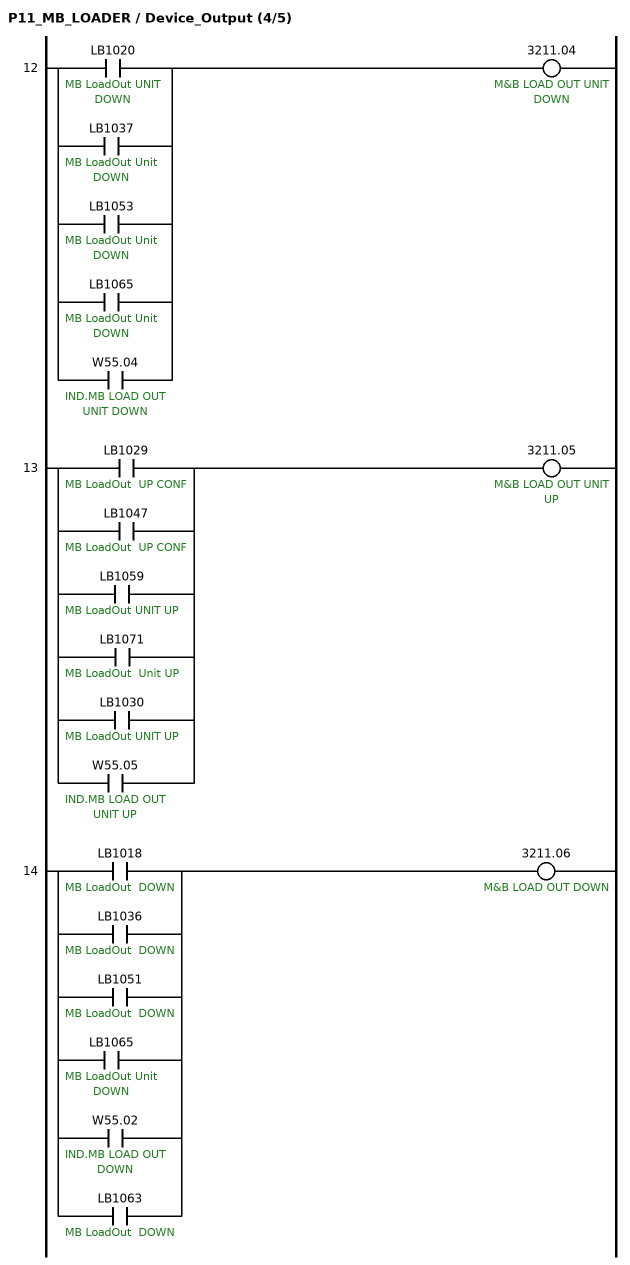
; [picture p144: P11_MB_LOADER / Device_Output, rungs 12-14]
; rung 12
LD LB1020  ; MB LoadOut UNIT DOWN
OR LB1037  ; MB LoadOut Unit  DOWN
OR LB1053  ; MB LoadOut Unit DOWN
OR LB1065  ; MB LoadOut Unit  DOWN
OR W55.04  ; IND.MB LOAD OUT UNIT DOWN
OUT 3211.04  ; M&B LOAD OUT UNIT DOWN
; rung 13
LD LB1029  ; MB LoadOut  UP CONF
OR LB1047  ; MB LoadOut  UP CONF
OR LB1059  ; MB LoadOut UNIT UP
OR LB1071  ; MB LoadOut  Unit UP
OR LB1030  ; MB LoadOut UNIT UP
OR W55.05  ; IND.MB LOAD OUT UNIT UP
OUT 3211.05  ; M&B LOAD OUT UNIT UP
; rung 14
LD LB1018  ; MB LoadOut  DOWN
OR LB1036  ; MB LoadOut  DOWN
OR LB1051  ; MB LoadOut  DOWN
OR LB1065  ; MB LoadOut Unit  DOWN
OR W55.02  ; IND.MB LOAD OUT DOWN
OR LB1063  ; MB LoadOut  DOWN
OUT 3211.06  ; M&B LOAD OUT DOWN

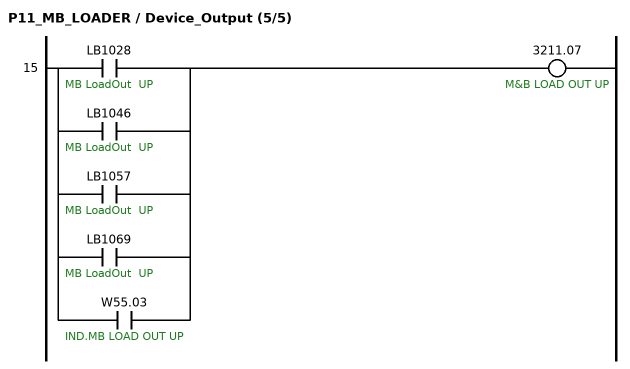
; rung 15
LD LB1028  ; MB LoadOut  UP
OR LB1046  ; MB LoadOut  UP
OR LB1057  ; MB LoadOut  UP
OR LB1069  ; MB LoadOut  UP
OR W55.03  ; IND.MB LOAD OUT UP
OUT 3211.07  ; M&B LOAD OUT UP

### Section Station_Output

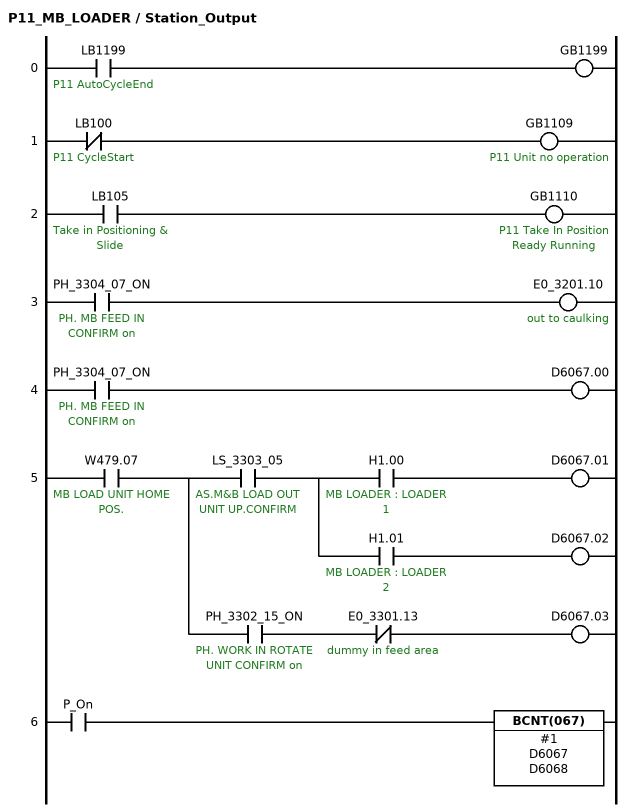
; rung 0
LD LB1199  ; P11 AutoCycleEnd
OUT GB1199
; rung 1
LDNOT LB100  ; P11 CycleStart
OUT GB1109  ; P11 Unit no operation
; rung 2
LD LB105  ; Take in Positioning & Slide
OUT GB1110  ; P11 Take In Position Ready Running
; rung 3
LD PH_3304_07_ON  ; PH. MB FEED IN CONFIRM on
OUT E0_3201.10  ; out to caulking
; rung 4
LD PH_3304_07_ON  ; PH. MB FEED IN CONFIRM on
OUT D6067.00
; rung 5
LD W479.07  ; MB LOAD UNIT HOME POS.
OUT TR0
AND LS_3303_05  ; AS.M&B LOAD OUT UNIT UP.CONFIRM
OUT TR1
AND H1.00  ; MB LOADER : LOADER 1
OUT D6067.01
LD TR1
AND H1.01  ; MB LOADER : LOADER 2
OUT D6067.02
LD TR0
AND PH_3302_15_ON  ; PH. WORK IN ROTATE UNIT CONFIRM on
ANDNOT E0_3301.13  ; dummy in feed area
OUT D6067.03
; rung 6
LD P_On
BCNT(067) #1 D6067 D6068

### Section Individual

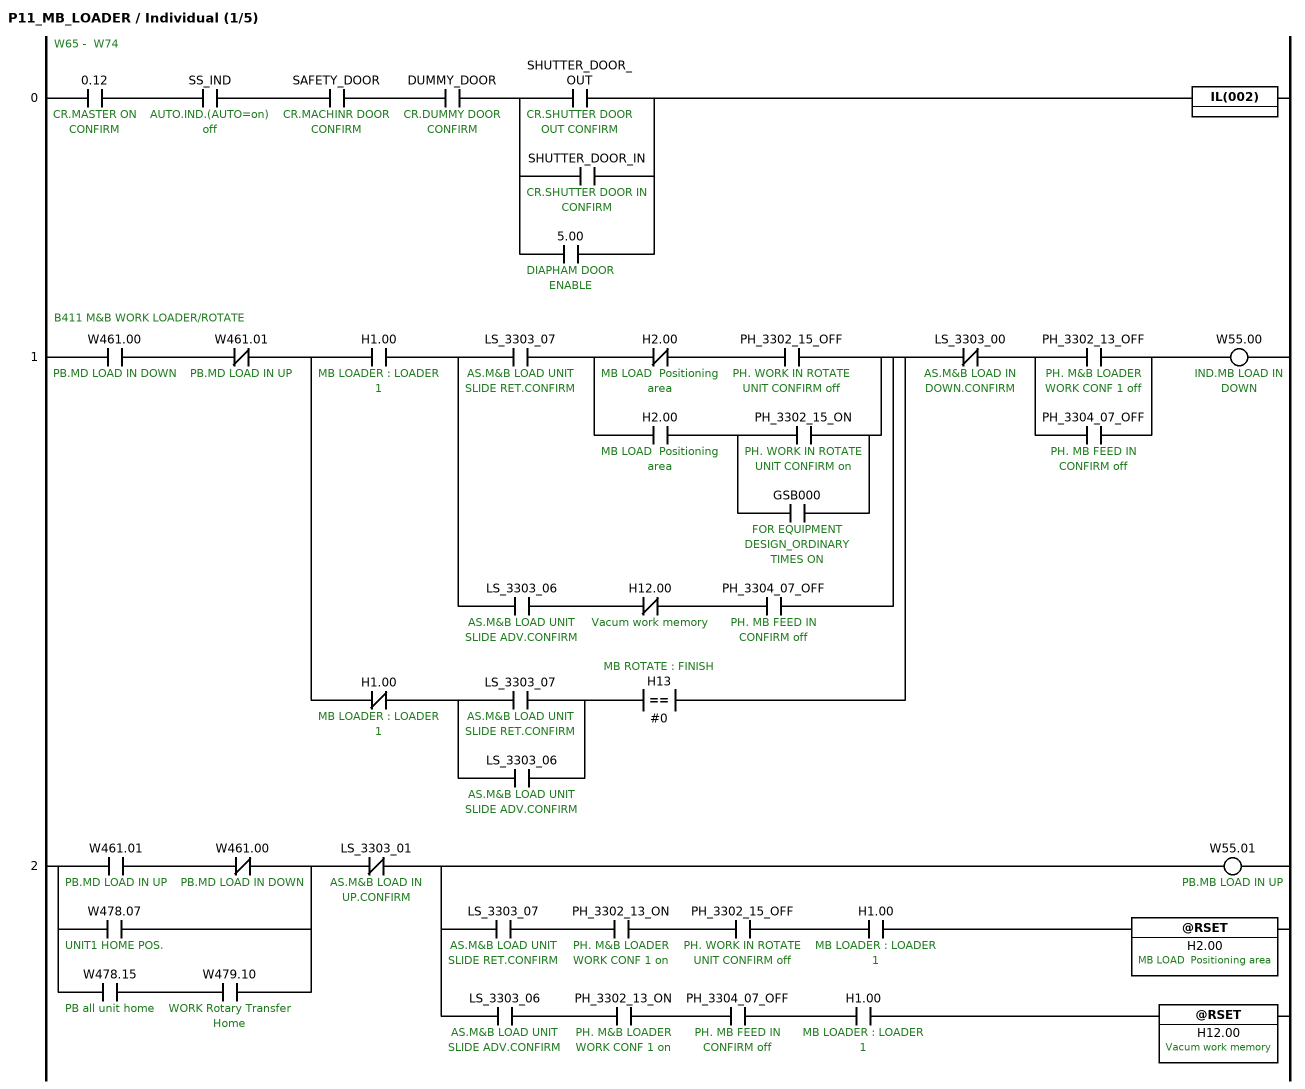
; rung 0: W65 -  W74
LD 0.12  ; CR.MASTER ON CONFIRM
AND SS_IND  ; AUTO.IND.(AUTO=on) off
AND SAFETY_DOOR  ; CR.MACHINR DOOR CONFIRM
AND DUMMY_DOOR  ; CR.DUMMY DOOR CONFIRM
LD SHUTTER_DOOR_OUT  ; CR.SHUTTER DOOR OUT CONFIRM
OR SHUTTER_DOOR_IN  ; CR.SHUTTER DOOR IN CONFIRM
OR 5.00  ; DIAPHAM DOOR ENABLE
ANDLD
IL(002)
; rung 1: B411 M&B WORK LOADER/ROTATE
LD W461.00  ; PB.MD LOAD IN DOWN
ANDNOT W461.01  ; PB.MD LOAD IN UP
LD H1.00  ; MB LOADER : LOADER 1
LD LS_3303_07  ; AS.M&B LOAD UNIT SLIDE RET.CONFIRM
LDNOT H2.00  ; MB LOAD  Positioning area
AND PH_3302_15_OFF  ; PH. WORK IN ROTATE UNIT CONFIRM off
LD H2.00  ; MB LOAD  Positioning area
LD PH_3302_15_ON  ; PH. WORK IN ROTATE UNIT CONFIRM on
OR GSB000  ; FOR EQUIPMENT DESIGN_ORDINARY TIMES ON
ANDLD
ORLD
ANDLD
LD LS_3303_06  ; AS.M&B LOAD UNIT SLIDE ADV.CONFIRM
ANDNOT H12.00  ; Vacum work memory
AND PH_3304_07_OFF  ; PH. MB FEED IN CONFIRM off
ORLD
ANDLD
LDNOT H1.00  ; MB LOADER : LOADER 1
LD LS_3303_07  ; AS.M&B LOAD UNIT SLIDE RET.CONFIRM
OR LS_3303_06  ; AS.M&B LOAD UNIT SLIDE ADV.CONFIRM
ANDLD
AND=(300) H13 #0  ; MB ROTATE : FINISH
ORLD
ANDLD
ANDNOT LS_3303_00  ; AS.M&B LOAD IN DOWN.CONFIRM
LD PH_3302_13_OFF  ; PH. M&B LOADER WORK CONF 1 off
OR PH_3304_07_OFF  ; PH. MB FEED IN CONFIRM off
ANDLD
OUT W55.00  ; IND.MB LOAD IN DOWN
; rung 2
LD W461.01  ; PB.MD LOAD IN UP
ANDNOT W461.00  ; PB.MD LOAD IN DOWN
OR W478.07  ; UNIT1 HOME POS.
LD W478.15  ; PB all unit home
AND W479.10  ; WORK Rotary Transfer Home
ORLD
ANDNOT LS_3303_01  ; AS.M&B LOAD IN UP.CONFIRM
OUT TR0
OUT W55.01  ; PB.MB LOAD IN UP
AND LS_3303_07  ; AS.M&B LOAD UNIT SLIDE RET.CONFIRM
AND PH_3302_13_ON  ; PH. M&B LOADER WORK CONF 1 on
AND PH_3302_15_OFF  ; PH. WORK IN ROTATE UNIT CONFIRM off
AND H1.00  ; MB LOADER : LOADER 1
@RSET H2.00  ; MB LOAD  Positioning area
LD TR0
AND LS_3303_06  ; AS.M&B LOAD UNIT SLIDE ADV.CONFIRM
AND PH_3302_13_ON  ; PH. M&B LOADER WORK CONF 1 on
AND PH_3304_07_OFF  ; PH. MB FEED IN CONFIRM off
AND H1.00  ; MB LOADER : LOADER 1
@RSET H12.00  ; Vacum work memory

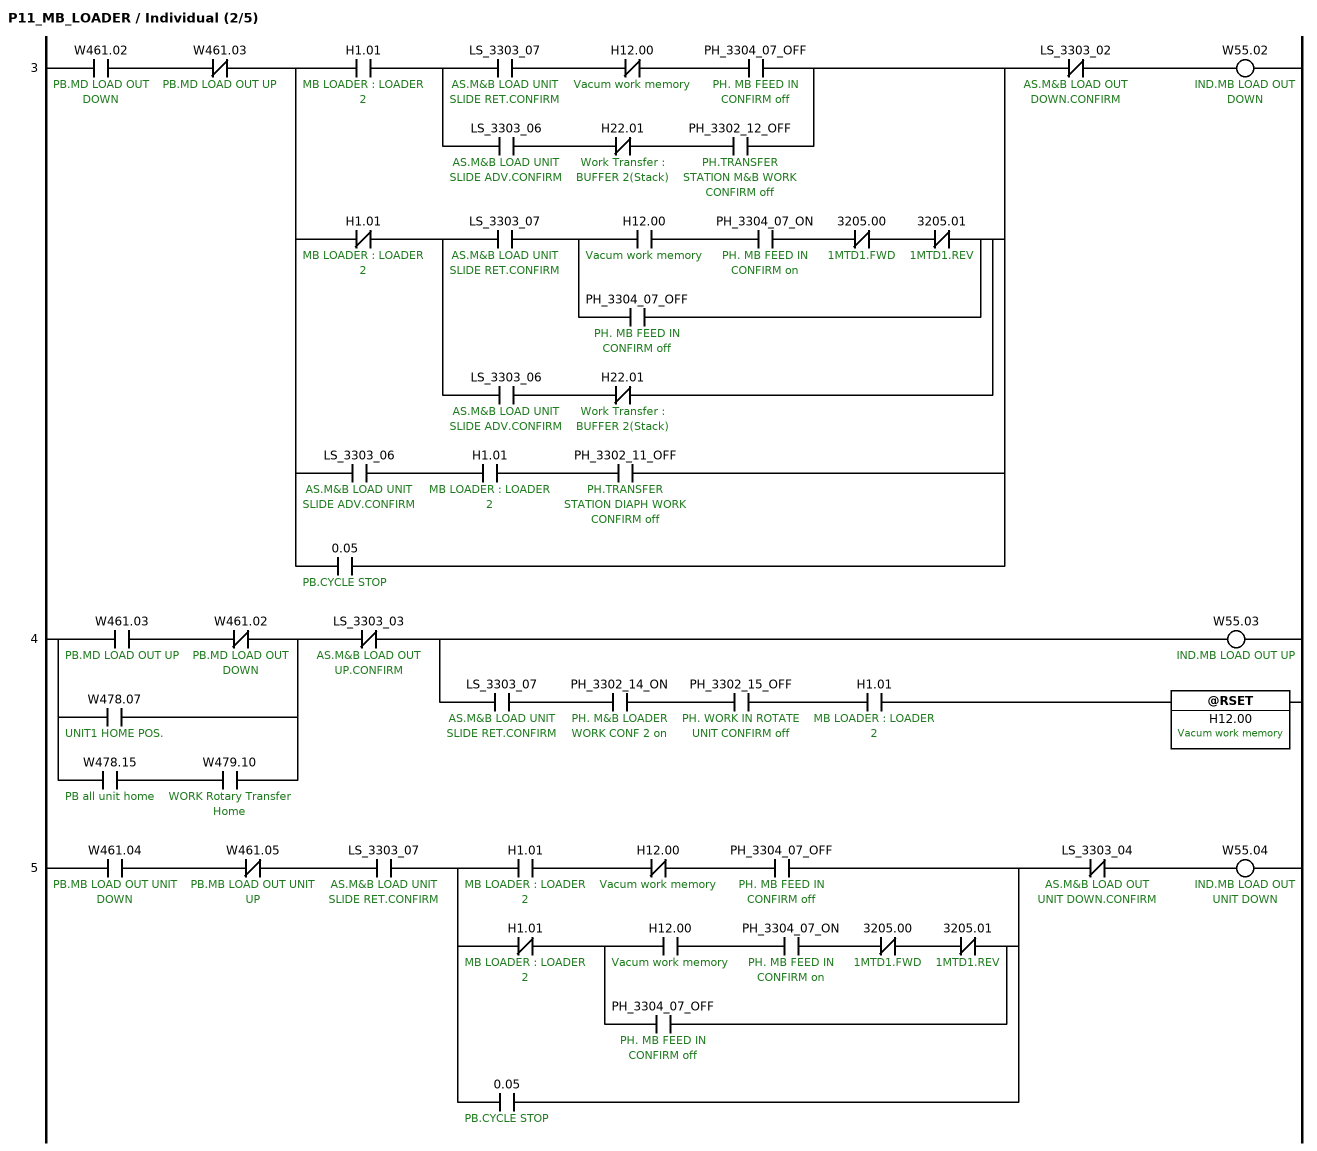
; rung 3
LD W461.02  ; PB.MD LOAD OUT DOWN
ANDNOT W461.03  ; PB.MD LOAD OUT UP
LD H1.01  ; MB LOADER : LOADER 2
LD LS_3303_07  ; AS.M&B LOAD UNIT SLIDE RET.CONFIRM
ANDNOT H12.00  ; Vacum work memory
AND PH_3304_07_OFF  ; PH. MB FEED IN CONFIRM off
LD LS_3303_06  ; AS.M&B LOAD UNIT SLIDE ADV.CONFIRM
ANDNOT H22.01  ; Work Transfer : BUFFER 2(Stack)
AND PH_3302_12_OFF  ; PH.TRANSFER STATION M&B WORK CONFIRM off
ORLD
ANDLD
LDNOT H1.01  ; MB LOADER : LOADER 2
LD LS_3303_07  ; AS.M&B LOAD UNIT SLIDE RET.CONFIRM
LD H12.00  ; Vacum work memory
AND PH_3304_07_ON  ; PH. MB FEED IN CONFIRM on
ANDNOT 3205.00  ; 1MTD1.FWD
ANDNOT 3205.01  ; 1MTD1.REV
OR PH_3304_07_OFF  ; PH. MB FEED IN CONFIRM off
ANDLD
LD LS_3303_06  ; AS.M&B LOAD UNIT SLIDE ADV.CONFIRM
ANDNOT H22.01  ; Work Transfer : BUFFER 2(Stack)  // Prohibit DOWN AFTER POSITIONING
ORLD
ANDLD
ORLD
LD LS_3303_06  ; AS.M&B LOAD UNIT SLIDE ADV.CONFIRM
AND H1.01  ; MB LOADER : LOADER 2
AND PH_3302_11_OFF  ; PH.TRANSFER STATION DIAPH WORK CONFIRM off
ORLD
OR 0.05  ; PB.CYCLE STOP
ANDLD
ANDNOT LS_3303_02  ; AS.M&B LOAD OUT DOWN.CONFIRM
OUT W55.02  ; IND.MB LOAD OUT DOWN
; rung 4
LD W461.03  ; PB.MD LOAD OUT UP
ANDNOT W461.02  ; PB.MD LOAD OUT DOWN
OR W478.07  ; UNIT1 HOME POS.
LD W478.15  ; PB all unit home
AND W479.10  ; WORK Rotary Transfer Home
ORLD
ANDNOT LS_3303_03  ; AS.M&B LOAD OUT UP.CONFIRM
OUT W55.03  ; IND.MB LOAD OUT UP
AND LS_3303_07  ; AS.M&B LOAD UNIT SLIDE RET.CONFIRM
AND PH_3302_14_ON  ; PH. M&B LOADER WORK CONF 2 on
AND PH_3302_15_OFF  ; PH. WORK IN ROTATE UNIT CONFIRM off
AND H1.01  ; MB LOADER : LOADER 2
@RSET H12.00  ; Vacum work memory
; rung 5
LD W461.04  ; PB.MB LOAD OUT UNIT DOWN
ANDNOT W461.05  ; PB.MB LOAD OUT UNIT UP
AND LS_3303_07  ; AS.M&B LOAD UNIT SLIDE RET.CONFIRM
LD H1.01  ; MB LOADER : LOADER 2
ANDNOT H12.00  ; Vacum work memory
AND PH_3304_07_OFF  ; PH. MB FEED IN CONFIRM off
LDNOT H1.01  ; MB LOADER : LOADER 2
LD H12.00  ; Vacum work memory
AND PH_3304_07_ON  ; PH. MB FEED IN CONFIRM on
ANDNOT 3205.00  ; 1MTD1.FWD
ANDNOT 3205.01  ; 1MTD1.REV
OR PH_3304_07_OFF  ; PH. MB FEED IN CONFIRM off
ANDLD
ORLD
OR 0.05  ; PB.CYCLE STOP
ANDLD
ANDNOT LS_3303_04  ; AS.M&B LOAD OUT UNIT DOWN.CONFIRM
OUT W55.04  ; IND.MB LOAD OUT UNIT DOWN

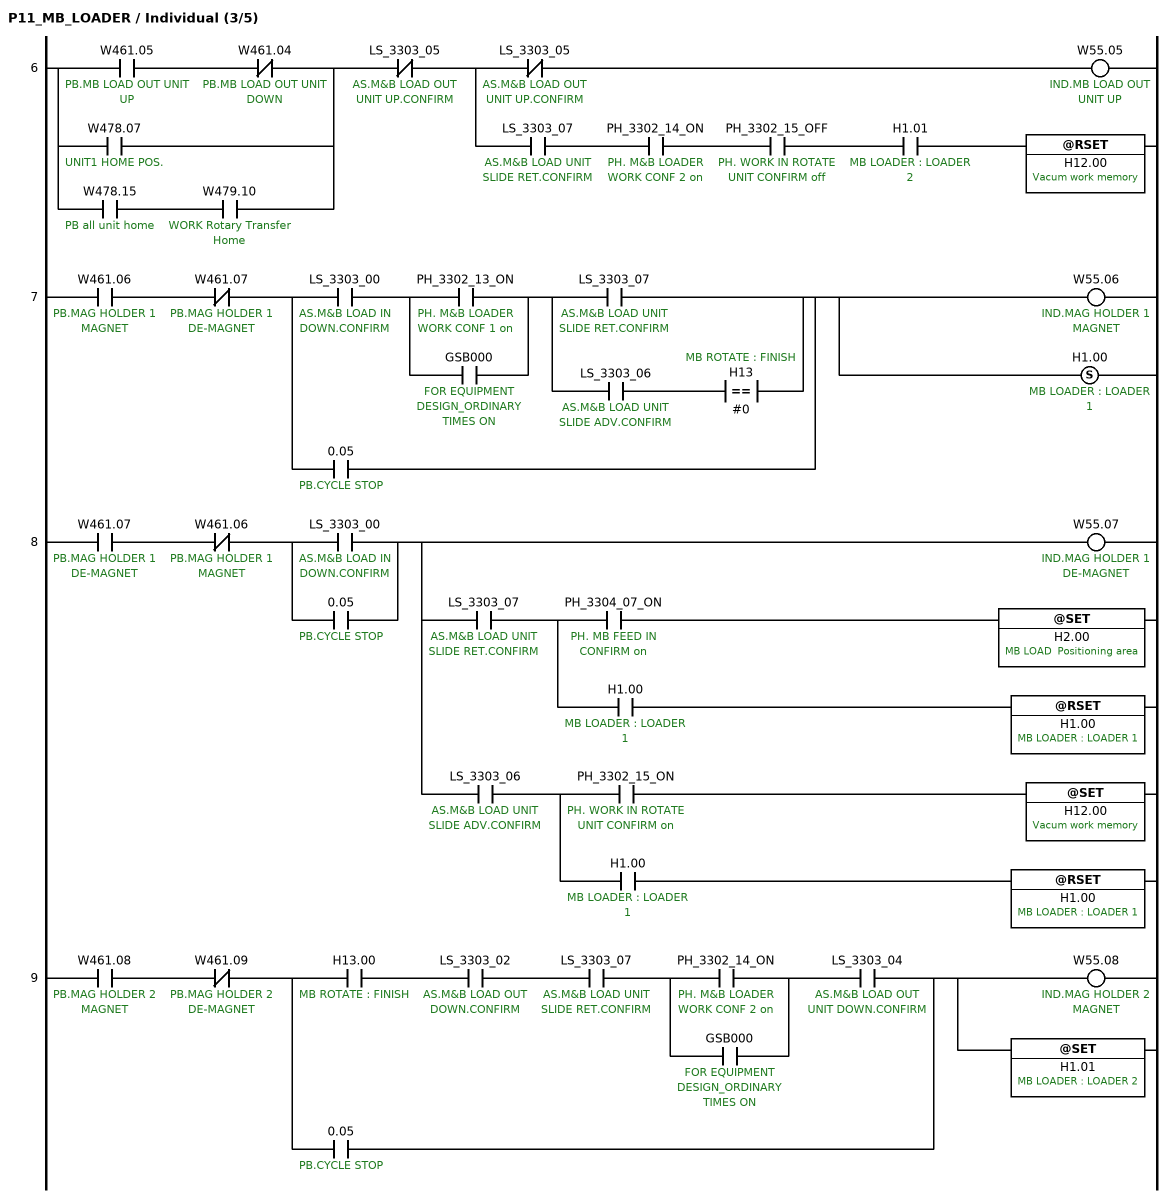
; rung 6
LD W461.05  ; PB.MB LOAD OUT UNIT UP
ANDNOT W461.04  ; PB.MB LOAD OUT UNIT DOWN
OR W478.07  ; UNIT1 HOME POS.
LD W478.15  ; PB all unit home
AND W479.10  ; WORK Rotary Transfer Home
ORLD
ANDNOT LS_3303_05  ; AS.M&B LOAD OUT UNIT UP.CONFIRM
OUT TR0
ANDNOT LS_3303_05  ; AS.M&B LOAD OUT UNIT UP.CONFIRM
OUT W55.05  ; IND.MB LOAD OUT UNIT UP
LD TR0
AND LS_3303_07  ; AS.M&B LOAD UNIT SLIDE RET.CONFIRM
AND PH_3302_14_ON  ; PH. M&B LOADER WORK CONF 2 on
AND PH_3302_15_OFF  ; PH. WORK IN ROTATE UNIT CONFIRM off
AND H1.01  ; MB LOADER : LOADER 2
@RSET H12.00  ; Vacum work memory
; rung 7
LD W461.06  ; PB.MAG HOLDER 1 MAGNET
ANDNOT W461.07  ; PB.MAG HOLDER 1 DE-MAGNET
LD LS_3303_00  ; AS.M&B LOAD IN DOWN.CONFIRM
LD PH_3302_13_ON  ; PH. M&B LOADER WORK CONF 1 on
OR GSB000  ; FOR EQUIPMENT DESIGN_ORDINARY TIMES ON
ANDLD
LD LS_3303_07  ; AS.M&B LOAD UNIT SLIDE RET.CONFIRM
LD LS_3303_06  ; AS.M&B LOAD UNIT SLIDE ADV.CONFIRM
AND=(300) H13 #0  ; MB ROTATE : FINISH
ORLD
ANDLD
OR 0.05  ; PB.CYCLE STOP
ANDLD
OUT W55.06  ; IND.MAG HOLDER 1 MAGNET
SET H1.00  ; MB LOADER : LOADER 1
; rung 8
LD W461.07  ; PB.MAG HOLDER 1 DE-MAGNET
ANDNOT W461.06  ; PB.MAG HOLDER 1 MAGNET
LD LS_3303_00  ; AS.M&B LOAD IN DOWN.CONFIRM
OR 0.05  ; PB.CYCLE STOP
ANDLD
OUT TR0
OUT W55.07  ; IND.MAG HOLDER 1 DE-MAGNET
AND LS_3303_07  ; AS.M&B LOAD UNIT SLIDE RET.CONFIRM
OUT TR1
AND PH_3304_07_ON  ; PH. MB FEED IN CONFIRM on
@SET H2.00  ; MB LOAD  Positioning area
LD TR1
AND H1.00  ; MB LOADER : LOADER 1
@RSET H1.00  ; MB LOADER : LOADER 1
LD TR0
AND LS_3303_06  ; AS.M&B LOAD UNIT SLIDE ADV.CONFIRM
OUT TR0
AND PH_3302_15_ON  ; PH. WORK IN ROTATE UNIT CONFIRM on
@SET H12.00  ; Vacum work memory
LD TR0
AND H1.00  ; MB LOADER : LOADER 1
@RSET H1.00  ; MB LOADER : LOADER 1
; rung 9
LD W461.08  ; PB.MAG HOLDER 2 MAGNET
ANDNOT W461.09  ; PB.MAG HOLDER 2 DE-MAGNET
LD H13.00  ; MB ROTATE : FINISH
AND LS_3303_02  ; AS.M&B LOAD OUT DOWN.CONFIRM
AND LS_3303_07  ; AS.M&B LOAD UNIT SLIDE RET.CONFIRM
LD PH_3302_14_ON  ; PH. M&B LOADER WORK CONF 2 on
OR GSB000  ; FOR EQUIPMENT DESIGN_ORDINARY TIMES ON
ANDLD
AND LS_3303_04  ; AS.M&B LOAD OUT UNIT DOWN.CONFIRM
OR 0.05  ; PB.CYCLE STOP
ANDLD
OUT W55.08  ; IND.MAG HOLDER 2 MAGNET  // PROHIBIT MAGNETIZE AFTER POSITIONING
@SET H1.01  ; MB LOADER : LOADER 2

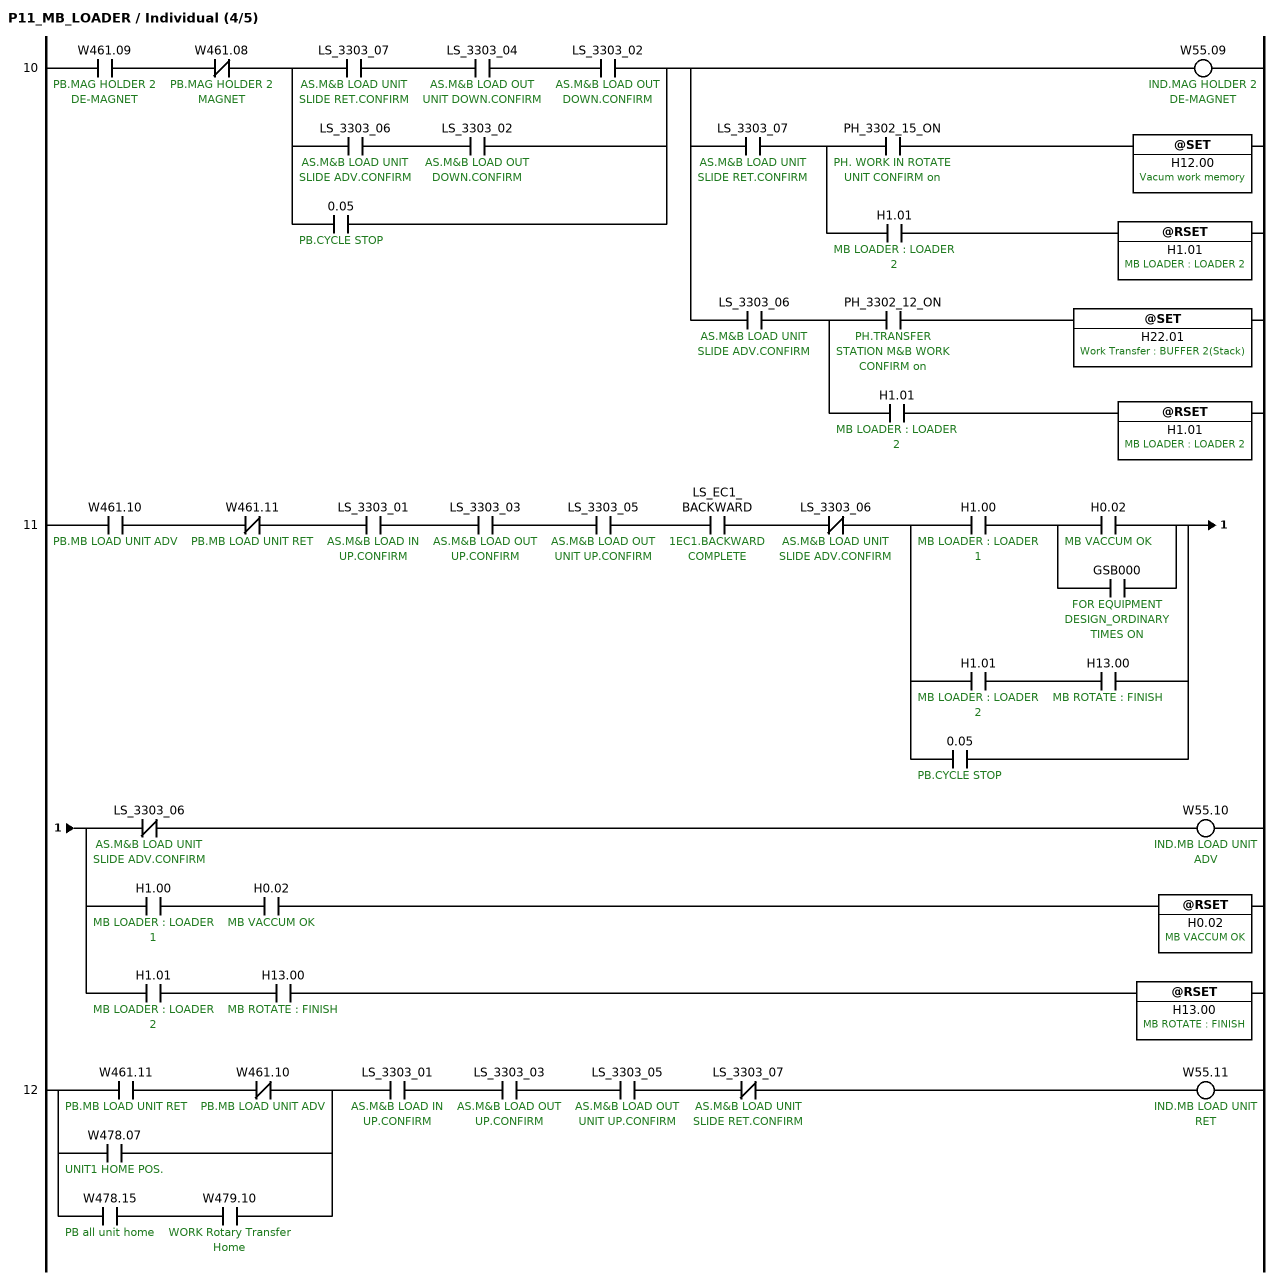
; rung 10
LD W461.09  ; PB.MAG HOLDER 2 DE-MAGNET
ANDNOT W461.08  ; PB.MAG HOLDER 2 MAGNET
LD LS_3303_07  ; AS.M&B LOAD UNIT SLIDE RET.CONFIRM
AND LS_3303_04  ; AS.M&B LOAD OUT UNIT DOWN.CONFIRM
AND LS_3303_02  ; AS.M&B LOAD OUT DOWN.CONFIRM
LD LS_3303_06  ; AS.M&B LOAD UNIT SLIDE ADV.CONFIRM
AND LS_3303_02  ; AS.M&B LOAD OUT DOWN.CONFIRM
ORLD
OR 0.05  ; PB.CYCLE STOP
ANDLD
OUT TR0
OUT W55.09  ; IND.MAG HOLDER 2 DE-MAGNET
AND LS_3303_07  ; AS.M&B LOAD UNIT SLIDE RET.CONFIRM
OUT TR1
AND PH_3302_15_ON  ; PH. WORK IN ROTATE UNIT CONFIRM on
@SET H12.00  ; Vacum work memory
LD TR1
AND H1.01  ; MB LOADER : LOADER 2
@RSET H1.01  ; MB LOADER : LOADER 2
LD TR0
AND LS_3303_06  ; AS.M&B LOAD UNIT SLIDE ADV.CONFIRM
OUT TR0
AND PH_3302_12_ON  ; PH.TRANSFER STATION M&B WORK CONFIRM on
@SET H22.01  ; Work Transfer : BUFFER 2(Stack)
LD TR0
AND H1.01  ; MB LOADER : LOADER 2
@RSET H1.01  ; MB LOADER : LOADER 2
; rung 11
LD W461.10  ; PB.MB LOAD UNIT ADV
ANDNOT W461.11  ; PB.MB LOAD UNIT RET
AND LS_3303_01  ; AS.M&B LOAD IN UP.CONFIRM
AND LS_3303_03  ; AS.M&B LOAD OUT UP.CONFIRM
AND LS_3303_05  ; AS.M&B LOAD OUT UNIT UP.CONFIRM
AND LS_EC1_BACKWARD  ; 1EC1.BACKWARD COMPLETE
ANDNOT LS_3303_06  ; AS.M&B LOAD UNIT SLIDE ADV.CONFIRM
LD H1.00  ; MB LOADER : LOADER 1
LD H0.02  ; MB VACCUM OK
OR GSB000  ; FOR EQUIPMENT DESIGN_ORDINARY TIMES ON
ANDLD
LD H1.01  ; MB LOADER : LOADER 2
AND H13.00  ; MB ROTATE : FINISH
ORLD
OR 0.05  ; PB.CYCLE STOP
ANDLD
OUT TR0
ANDNOT LS_3303_06  ; AS.M&B LOAD UNIT SLIDE ADV.CONFIRM
OUT W55.10  ; IND.MB LOAD UNIT ADV
LD TR0
AND H1.00  ; MB LOADER : LOADER 1
AND H0.02  ; MB VACCUM OK
@RSET H0.02  ; MB VACCUM OK
LD TR0
AND H1.01  ; MB LOADER : LOADER 2
AND H13.00  ; MB ROTATE : FINISH
@RSET H13.00  ; MB ROTATE : FINISH
; rung 12
LD W461.11  ; PB.MB LOAD UNIT RET
ANDNOT W461.10  ; PB.MB LOAD UNIT ADV
OR W478.07  ; UNIT1 HOME POS.
LD W478.15  ; PB all unit home
AND W479.10  ; WORK Rotary Transfer Home
ORLD
AND LS_3303_01  ; AS.M&B LOAD IN UP.CONFIRM
AND LS_3303_03  ; AS.M&B LOAD OUT UP.CONFIRM
AND LS_3303_05  ; AS.M&B LOAD OUT UNIT UP.CONFIRM
ANDNOT LS_3303_07  ; AS.M&B LOAD UNIT SLIDE RET.CONFIRM
OUT W55.11  ; IND.MB LOAD UNIT RET

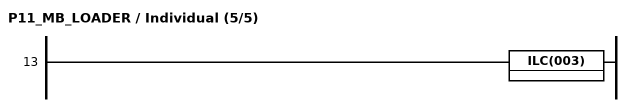
; rung 13
ILC(003)

### Section END
; rung 0
END(001)

## Program P12_MB_POSITIONING (cyclic task 2)
Local symbols
LB1199 E0_12.13 BOOL  ; P11 AutoCycleEnd
LB1200 E0_12.14 BOOL  ; AUTO START BEGIN
LB1201 E0_12.15 BOOL  ; WORK ROTATE START
LB1202 E0_13.00 BOOL  ; WORK ROTATE START 1CONF
LB1203 E0_13.01 BOOL  ; WORK ROTATE PIN UP
LB1204 E0_13.02 BOOL  ; WORK ROTATE PIN UP CONF
LB1205 E0_13.03 BOOL  ; MOTOR ROTATE SLOW DOWN
LB1206 E0_13.04 BOOL  ; MOTOR ROTATE STOP CONF
LB1210 E0_13.05 BOOL  ; AUTO START BEGIN
LB1211 E0_13.06 BOOL  ; WORK ROTATE PIN DOWN
LB1212 E0_13.07 BOOL  ; WORK ROTATE PIN DOWN CONF
LB1397 E0_13.08 BOOL  ; P12 AutoCycleEnd1
LB1398 E0_13.09 BOOL  ; P12 AutoCycleEnd2
LB1399 E0_13.10 BOOL  ; P12 AutoCycleEnd
LB200 E0_13.11 BOOL  ; P12 CycleStart
LB201 E0_13.12 BOOL  ; P12 ROTAE WORK
LB2010 E0_13.13 BOOL  ; SOL.GIPPER TRANSFER 2 CHUCK CONF
LB202 E0_13.14 BOOL  ; P12 ROTATE WORK DONE
LB340 E0_13.15 BOOL  ; IND 1 CYCLE
LB4543 E0_47.15 BOOL  ; dummy on magnet fall memory
LT209 T3029 TIMER

### Section HMI_Output

### Section Autorun

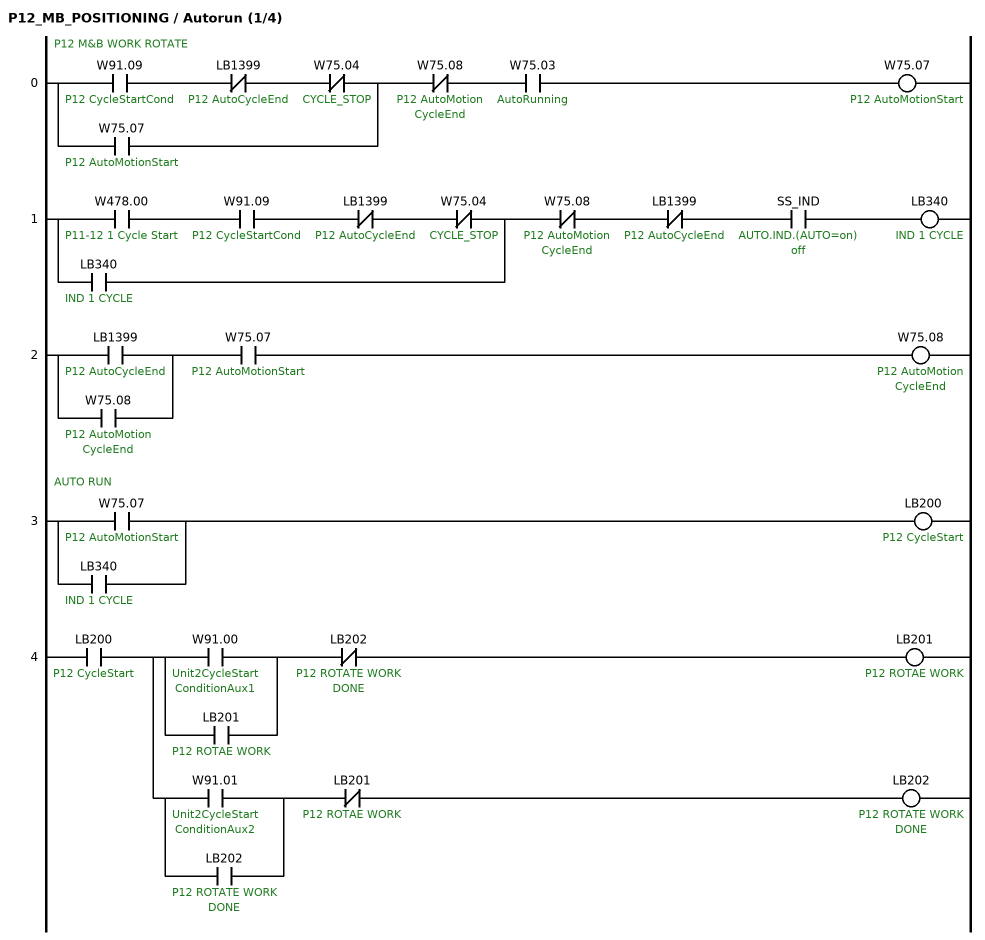
; rung 0: P12 M&B WORK ROTATE
LD W91.09  ; P12 CycleStartCond
ANDNOT LB1399  ; P12 AutoCycleEnd
ANDNOT W75.04  ; CYCLE_STOP
OR W75.07  ; P12 AutoMotionStart
ANDNOT W75.08  ; P12 AutoMotion CycleEnd
AND W75.03  ; AutoRunning
OUT W75.07  ; P12 AutoMotionStart
; rung 1
LD W478.00  ; P11-12 1 Cycle Start
AND W91.09  ; P12 CycleStartCond
ANDNOT LB1399  ; P12 AutoCycleEnd
ANDNOT W75.04  ; CYCLE_STOP
OR LB340  ; IND 1 CYCLE
ANDNOT W75.08  ; P12 AutoMotion CycleEnd
ANDNOT LB1399  ; P12 AutoCycleEnd
AND SS_IND  ; AUTO.IND.(AUTO=on) off
OUT LB340  ; IND 1 CYCLE
; rung 2
LD LB1399  ; P12 AutoCycleEnd
OR W75.08  ; P12 AutoMotion CycleEnd
AND W75.07  ; P12 AutoMotionStart
OUT W75.08  ; P12 AutoMotion CycleEnd
; rung 3: AUTO RUN
LD W75.07  ; P12 AutoMotionStart
OR LB340  ; IND 1 CYCLE
OUT LB200  ; P12 CycleStart
; rung 4
LD LB200  ; P12 CycleStart
OUT TR0
LD W91.00  ; Unit2CycleStartConditionAux1
OR LB201  ; P12 ROTAE WORK
ANDLD
ANDNOT LB202  ; P12 ROTATE WORK DONE
OUT LB201  ; P12 ROTAE WORK
LD TR0
LD W91.01  ; Unit2CycleStartConditionAux2
OR LB202  ; P12 ROTATE WORK DONE
ANDLD
ANDNOT LB201  ; P12 ROTAE WORK
OUT LB202  ; P12 ROTATE WORK DONE

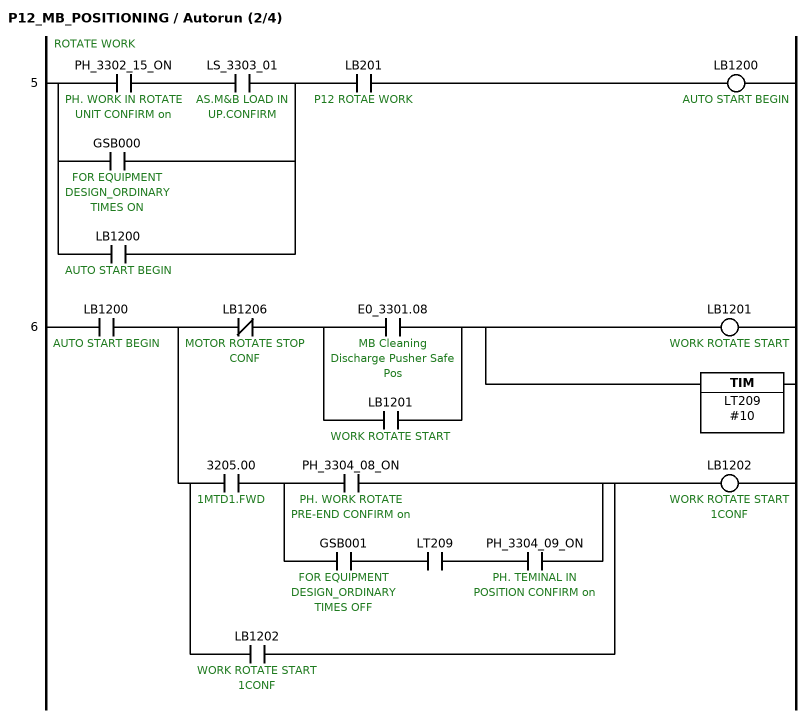
; rung 5: ROTATE WORK
LD PH_3302_15_ON  ; PH. WORK IN ROTATE UNIT CONFIRM on
AND LS_3303_01  ; AS.M&B LOAD IN UP.CONFIRM
OR GSB000  ; FOR EQUIPMENT DESIGN_ORDINARY TIMES ON
OR LB1200  ; AUTO START BEGIN
AND LB201  ; P12 ROTAE WORK
OUT LB1200  ; AUTO START BEGIN
; rung 6
LD LB1200  ; AUTO START BEGIN
OUT TR0
ANDNOT LB1206  ; MOTOR ROTATE STOP CONF
LD E0_3301.08  ; MB Cleaning Discharge Pusher Safe Pos
OR LB1201  ; WORK ROTATE START
ANDLD
OUT LB1201  ; WORK ROTATE START
TIM LT209 #10
LD TR0
LD 3205.00  ; 1MTD1.FWD
LD PH_3304_08_ON  ; PH. WORK ROTATE PRE-END CONFIRM on
LD GSB001  ; FOR EQUIPMENT DESIGN_ORDINARY TIMES OFF
AND LT209
AND PH_3304_09_ON  ; PH. TEMINAL IN POSITION CONFIRM on
ORLD
ANDLD
OR LB1202  ; WORK ROTATE START 1CONF
ANDLD
OUT LB1202  ; WORK ROTATE START 1CONF

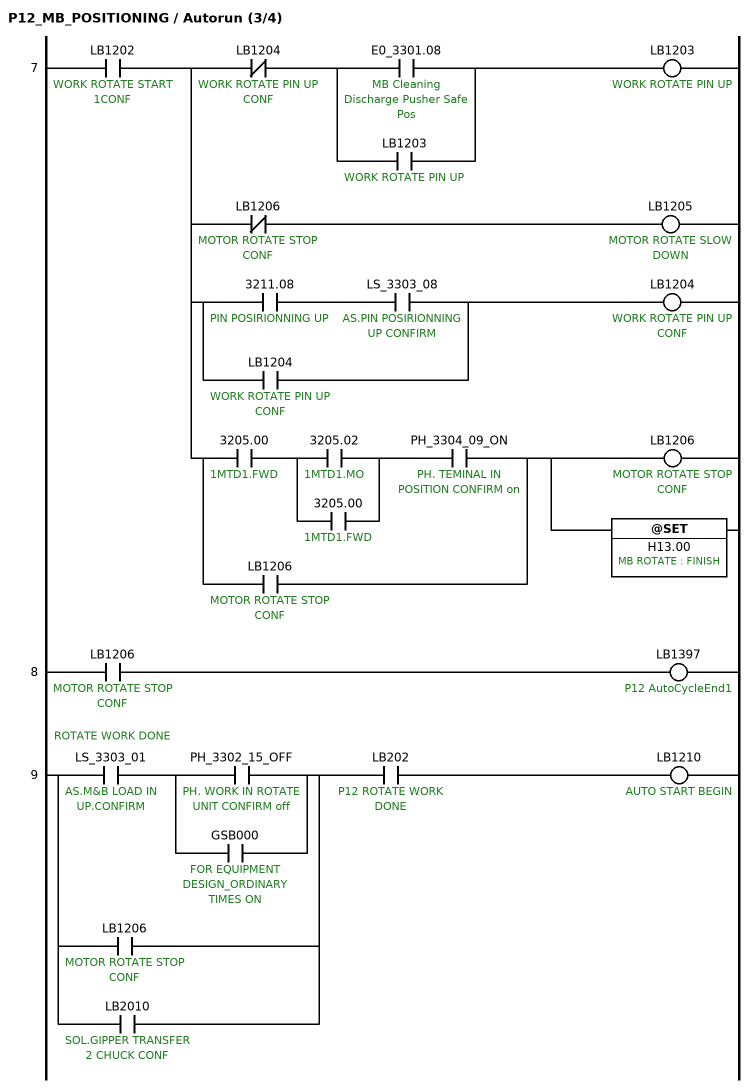
; rung 7
LD LB1202  ; WORK ROTATE START 1CONF
OUT TR0
ANDNOT LB1204  ; WORK ROTATE PIN UP CONF
LD E0_3301.08  ; MB Cleaning Discharge Pusher Safe Pos
OR LB1203  ; WORK ROTATE PIN UP
ANDLD
OUT LB1203  ; WORK ROTATE PIN UP
LD TR0
ANDNOT LB1206  ; MOTOR ROTATE STOP CONF
OUT LB1205  ; MOTOR ROTATE SLOW DOWN
LD TR0
LD 3211.08  ; PIN POSIRIONNING UP
AND LS_3303_08  ; AS.PIN POSIRIONNING UP CONFIRM
OR LB1204  ; WORK ROTATE PIN UP CONF
ANDLD
OUT LB1204  ; WORK ROTATE PIN UP CONF
LD TR0
LD 3205.00  ; 1MTD1.FWD
LD 3205.02  ; 1MTD1.MO
OR 3205.00  ; 1MTD1.FWD
ANDLD
AND PH_3304_09_ON  ; PH. TEMINAL IN POSITION CONFIRM on
OR LB1206  ; MOTOR ROTATE STOP CONF
ANDLD
OUT LB1206  ; MOTOR ROTATE STOP CONF
@SET H13.00  ; MB ROTATE : FINISH
; rung 8
LD LB1206  ; MOTOR ROTATE STOP CONF
OUT LB1397  ; P12 AutoCycleEnd1
; rung 9: ROTATE WORK DONE
LD LS_3303_01  ; AS.M&B LOAD IN UP.CONFIRM
LD PH_3302_15_OFF  ; PH. WORK IN ROTATE UNIT CONFIRM off
OR GSB000  ; FOR EQUIPMENT DESIGN_ORDINARY TIMES ON
ANDLD
OR LB1206  ; MOTOR ROTATE STOP CONF
OR LB2010  ; SOL.GIPPER TRANSFER 2 CHUCK CONF
AND LB202  ; P12 ROTATE WORK DONE
OUT LB1210  ; AUTO START BEGIN

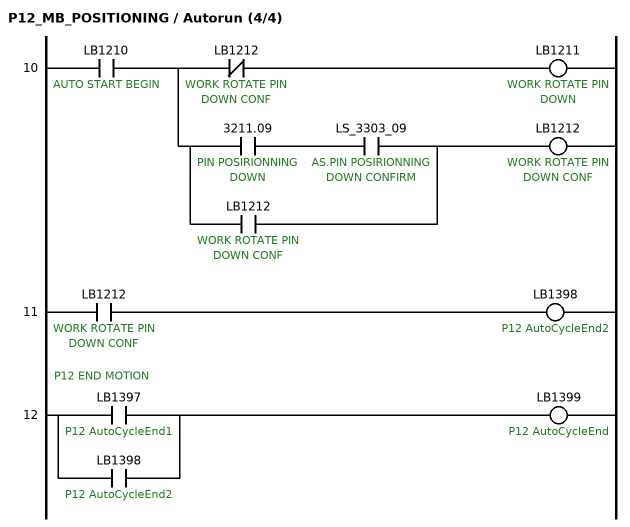
; rung 10
LD LB1210  ; AUTO START BEGIN
OUT TR0
ANDNOT LB1212  ; WORK ROTATE PIN DOWN CONF
OUT LB1211  ; WORK ROTATE PIN DOWN
LD TR0
LD 3211.09  ; PIN POSIRIONNING DOWN
AND LS_3303_09  ; AS.PIN POSIRIONNING DOWN CONFIRM
OR LB1212  ; WORK ROTATE PIN DOWN CONF
ANDLD
OUT LB1212  ; WORK ROTATE PIN DOWN CONF
; rung 11
LD LB1212  ; WORK ROTATE PIN DOWN CONF
OUT LB1398  ; P12 AutoCycleEnd2
; rung 12: P12 END MOTION
LD LB1397  ; P12 AutoCycleEnd1
OR LB1398  ; P12 AutoCycleEnd2
OUT LB1399  ; P12 AutoCycleEnd

### Section Condition

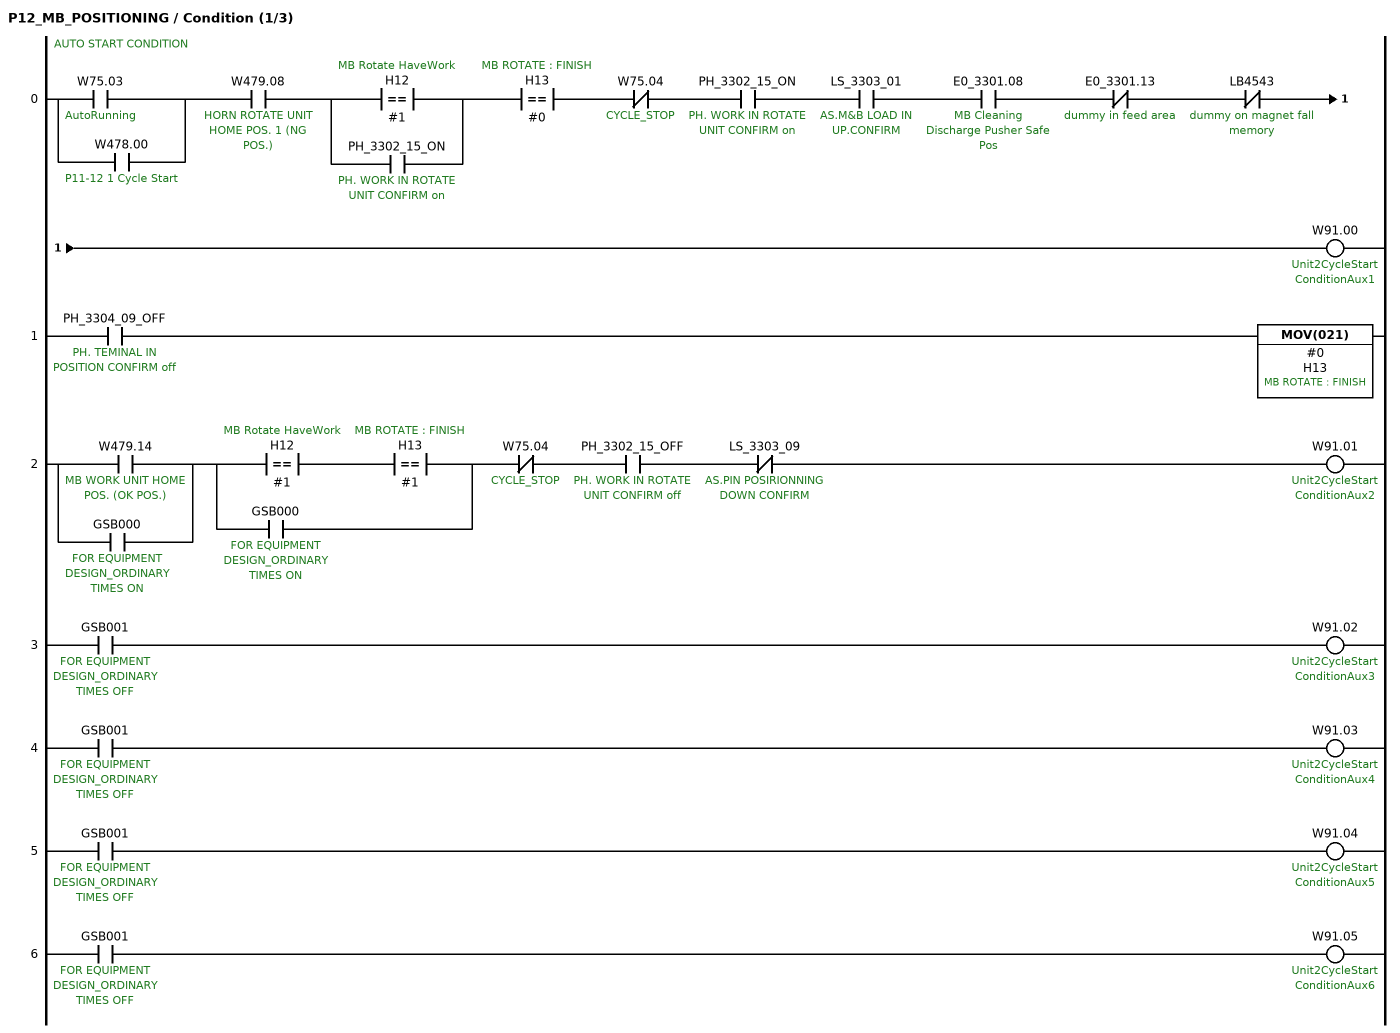
; rung 0: AUTO START CONDITION
LD W75.03  ; AutoRunning
OR W478.00  ; P11-12 1 Cycle Start
AND W479.08  ; HORN ROTATE UNIT HOME POS. 1 (NG POS.)
LD=(300) H12 #1  ; MB Rotate HaveWork
OR PH_3302_15_ON  ; PH. WORK IN ROTATE UNIT CONFIRM on
ANDLD
AND=(300) H13 #0  ; MB ROTATE : FINISH
ANDNOT W75.04  ; CYCLE_STOP
AND PH_3302_15_ON  ; PH. WORK IN ROTATE UNIT CONFIRM on
AND LS_3303_01  ; AS.M&B LOAD IN UP.CONFIRM
AND E0_3301.08  ; MB Cleaning Discharge Pusher Safe Pos
ANDNOT E0_3301.13  ; dummy in feed area
ANDNOT LB4543  ; dummy on magnet fall memory
OUT W91.00  ; Unit2CycleStartConditionAux1
; rung 1
LD PH_3304_09_OFF  ; PH. TEMINAL IN POSITION CONFIRM off
MOV(021) #0 H13  ; MB ROTATE : FINISH
; rung 2
LD W479.14  ; MB WORK UNIT HOME POS. (OK POS.)
OR GSB000  ; FOR EQUIPMENT DESIGN_ORDINARY TIMES ON
LD=(300) H12 #1  ; MB Rotate HaveWork
AND=(300) H13 #1  ; MB ROTATE : FINISH
OR GSB000  ; FOR EQUIPMENT DESIGN_ORDINARY TIMES ON
ANDLD
ANDNOT W75.04  ; CYCLE_STOP
AND PH_3302_15_OFF  ; PH. WORK IN ROTATE UNIT CONFIRM off
ANDNOT LS_3303_09  ; AS.PIN POSIRIONNING DOWN CONFIRM
OUT W91.01  ; Unit2CycleStartConditionAux2
; rung 3
LD GSB001  ; FOR EQUIPMENT DESIGN_ORDINARY TIMES OFF
OUT W91.02  ; Unit2CycleStartConditionAux3
; rung 4
LD GSB001  ; FOR EQUIPMENT DESIGN_ORDINARY TIMES OFF
OUT W91.03  ; Unit2CycleStartConditionAux4
; rung 5
LD GSB001  ; FOR EQUIPMENT DESIGN_ORDINARY TIMES OFF
OUT W91.04  ; Unit2CycleStartConditionAux5
; rung 6
LD GSB001  ; FOR EQUIPMENT DESIGN_ORDINARY TIMES OFF
OUT W91.05  ; Unit2CycleStartConditionAux6

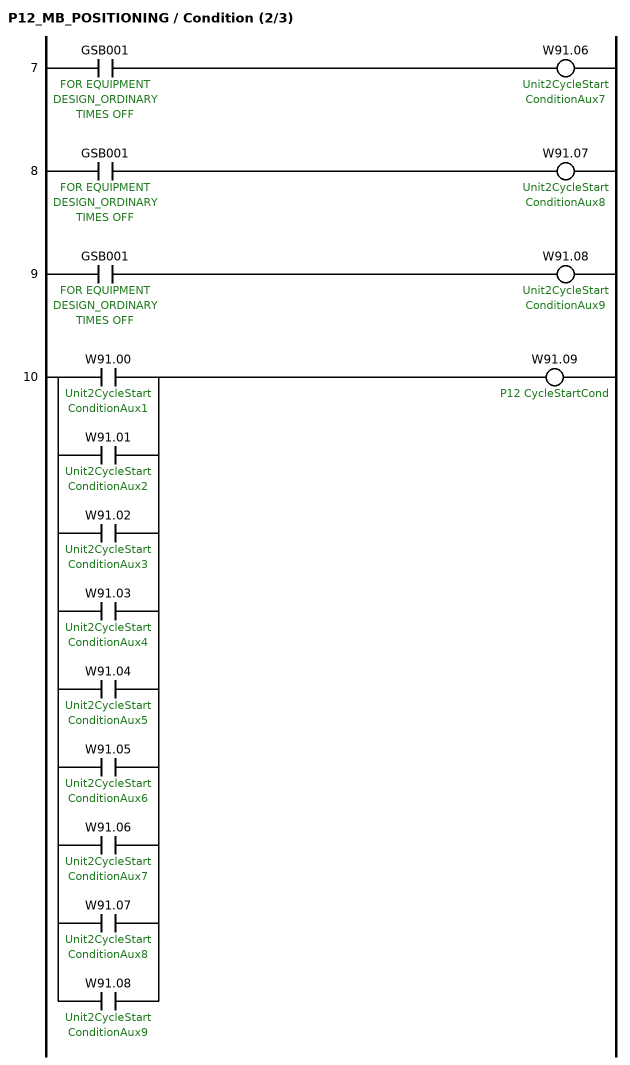
; rung 7
LD GSB001  ; FOR EQUIPMENT DESIGN_ORDINARY TIMES OFF
OUT W91.06  ; Unit2CycleStartConditionAux7
; rung 8
LD GSB001  ; FOR EQUIPMENT DESIGN_ORDINARY TIMES OFF
OUT W91.07  ; Unit2CycleStartConditionAux8
; rung 9
LD GSB001  ; FOR EQUIPMENT DESIGN_ORDINARY TIMES OFF
OUT W91.08  ; Unit2CycleStartConditionAux9
; rung 10
LD W91.00  ; Unit2CycleStartConditionAux1
OR W91.01  ; Unit2CycleStartConditionAux2
OR W91.02  ; Unit2CycleStartConditionAux3
OR W91.03  ; Unit2CycleStartConditionAux4
OR W91.04  ; Unit2CycleStartConditionAux5
OR W91.05  ; Unit2CycleStartConditionAux6
OR W91.06  ; Unit2CycleStartConditionAux7
OR W91.07  ; Unit2CycleStartConditionAux8
OR W91.08  ; Unit2CycleStartConditionAux9
OUT W91.09  ; P12 CycleStartCond

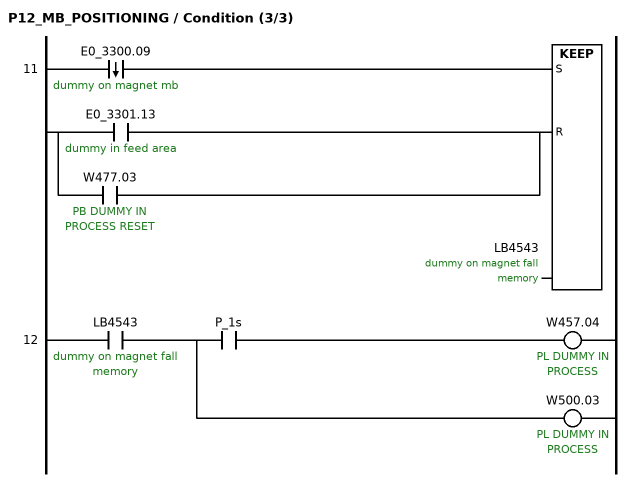
; rung 11
%LD E0_3300.09  ; dummy on magnet mb
LD E0_3301.13  ; dummy in feed area
OR W477.03  ; PB DUMMY IN PROCESS RESET
KEEP LB4543  ; dummy on magnet fall memory
; rung 12
LD LB4543  ; dummy on magnet fall memory
OUT TR0
AND P_1s
OUT W457.04  ; PL DUMMY IN PROCESS
LD TR0
OUT W500.03  ; PL DUMMY IN PROCESS

### Section Device_Output

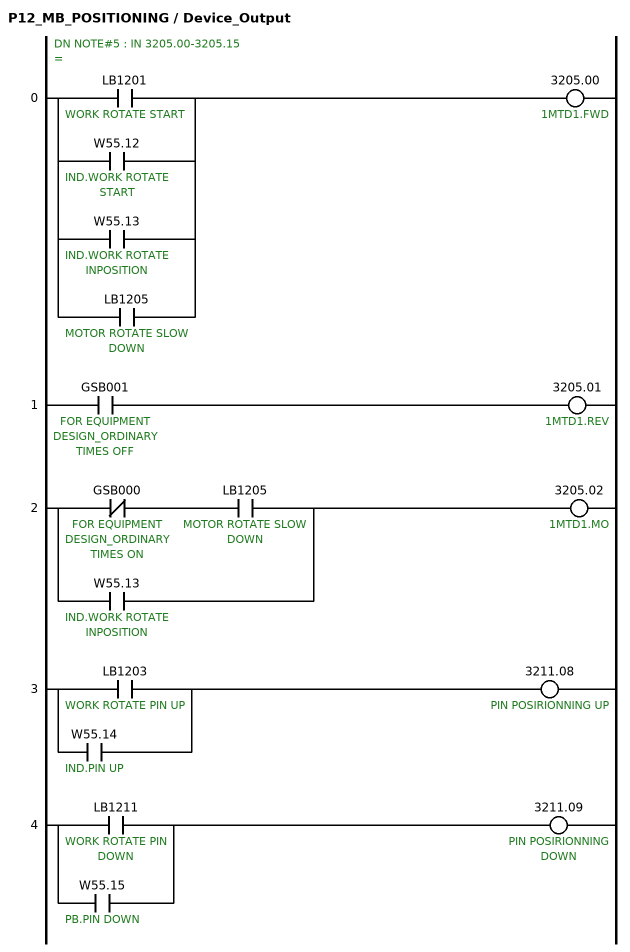
; rung 0: DN NOTE#5 : IN 3205.00-3205.15 / =
LD LB1201  ; WORK ROTATE START
OR W55.12  ; IND.WORK ROTATE START
OR W55.13  ; IND.WORK ROTATE INPOSITION
OR LB1205  ; MOTOR ROTATE SLOW DOWN
OUT 3205.00  ; 1MTD1.FWD
; rung 1
LD GSB001  ; FOR EQUIPMENT DESIGN_ORDINARY TIMES OFF
OUT 3205.01  ; 1MTD1.REV
; rung 2
LDNOT GSB000  ; FOR EQUIPMENT DESIGN_ORDINARY TIMES ON
AND LB1205  ; MOTOR ROTATE SLOW DOWN
OR W55.13  ; IND.WORK ROTATE INPOSITION
OUT 3205.02  ; 1MTD1.MO
; rung 3
LD LB1203  ; WORK ROTATE PIN UP
OR W55.14  ; IND.PIN UP
OUT 3211.08  ; PIN POSIRIONNING UP
; rung 4
LD LB1211  ; WORK ROTATE PIN DOWN
OR W55.15  ; PB.PIN DOWN
OUT 3211.09  ; PIN POSIRIONNING DOWN

### Section Station_Output

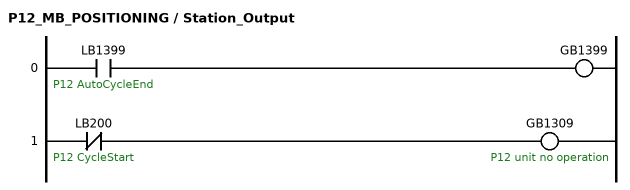
; rung 0
LD LB1399  ; P12 AutoCycleEnd
OUT GB1399
; rung 1
LDNOT LB200  ; P12 CycleStart
OUT GB1309  ; P12 unit no operation

### Section Individual

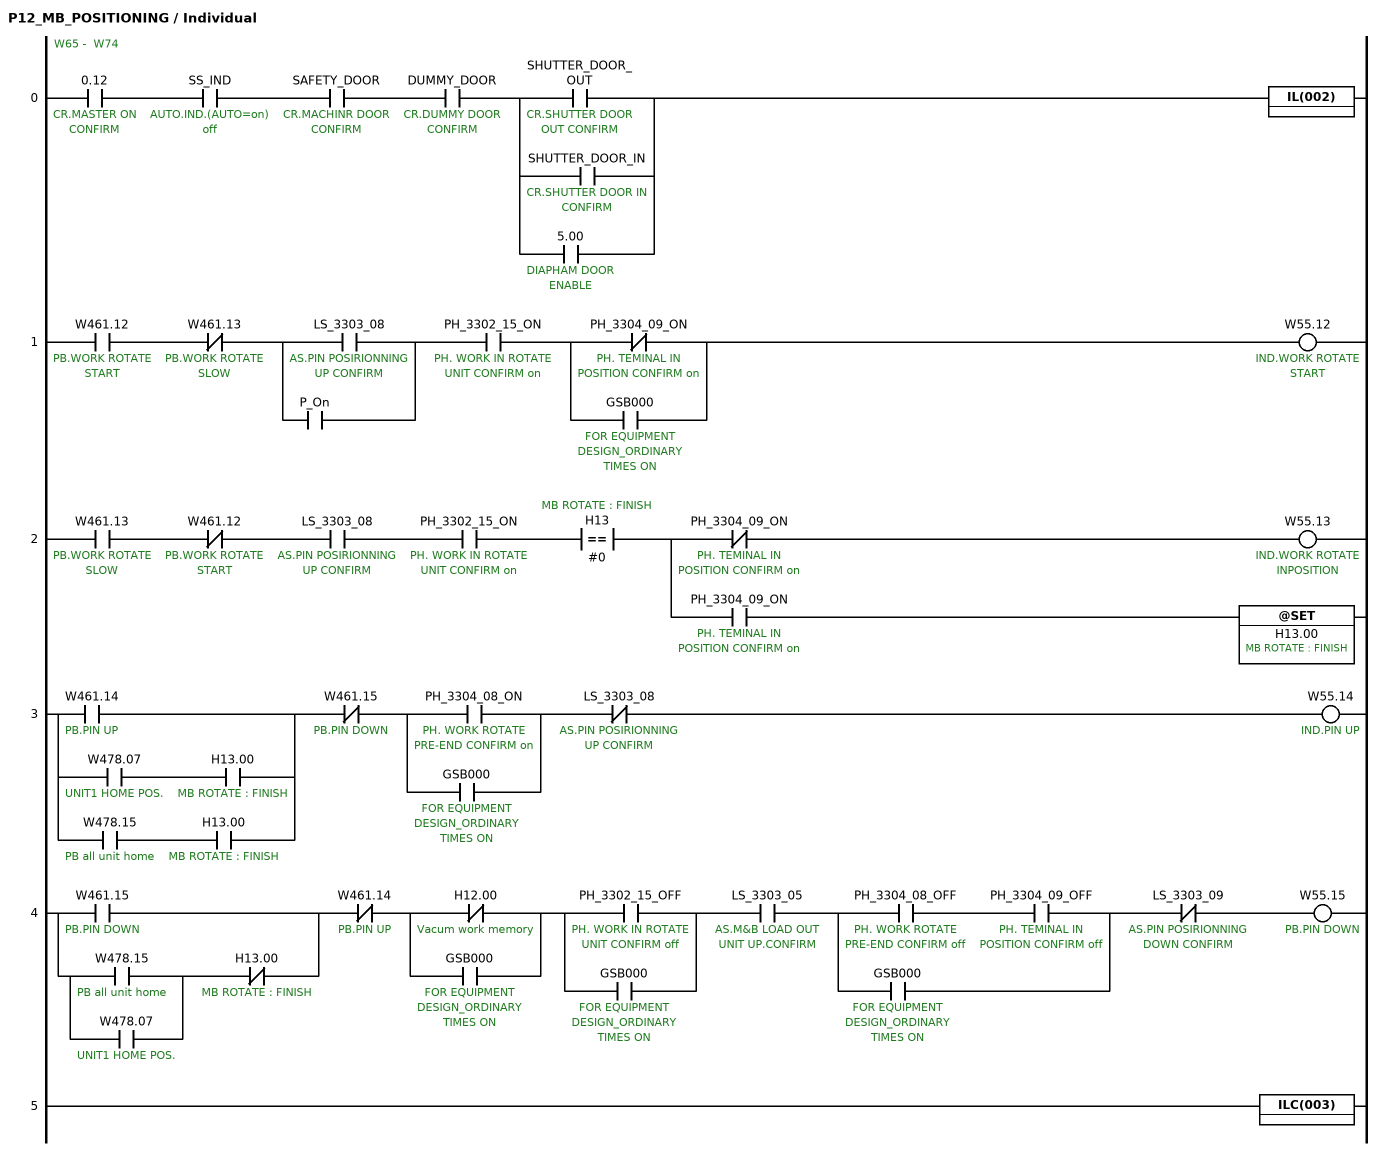
; rung 0: W65 -  W74
LD 0.12  ; CR.MASTER ON CONFIRM
AND SS_IND  ; AUTO.IND.(AUTO=on) off
AND SAFETY_DOOR  ; CR.MACHINR DOOR CONFIRM
AND DUMMY_DOOR  ; CR.DUMMY DOOR CONFIRM
LD SHUTTER_DOOR_OUT  ; CR.SHUTTER DOOR OUT CONFIRM
OR SHUTTER_DOOR_IN  ; CR.SHUTTER DOOR IN CONFIRM
OR 5.00  ; DIAPHAM DOOR ENABLE
ANDLD
IL(002)
; rung 1
LD W461.12  ; PB.WORK ROTATE START
ANDNOT W461.13  ; PB.WORK ROTATE SLOW
LD LS_3303_08  ; AS.PIN POSIRIONNING UP CONFIRM
OR P_On
ANDLD
AND PH_3302_15_ON  ; PH. WORK IN ROTATE UNIT CONFIRM on
LDNOT PH_3304_09_ON  ; PH. TEMINAL IN POSITION CONFIRM on
OR GSB000  ; FOR EQUIPMENT DESIGN_ORDINARY TIMES ON
ANDLD
OUT W55.12  ; IND.WORK ROTATE START
; rung 2
LD W461.13  ; PB.WORK ROTATE SLOW
ANDNOT W461.12  ; PB.WORK ROTATE START
AND LS_3303_08  ; AS.PIN POSIRIONNING UP CONFIRM
AND PH_3302_15_ON  ; PH. WORK IN ROTATE UNIT CONFIRM on
AND=(300) H13 #0  ; MB ROTATE : FINISH
OUT TR0
ANDNOT PH_3304_09_ON  ; PH. TEMINAL IN POSITION CONFIRM on
OUT W55.13  ; IND.WORK ROTATE INPOSITION
LD TR0
AND PH_3304_09_ON  ; PH. TEMINAL IN POSITION CONFIRM on
@SET H13.00  ; MB ROTATE : FINISH
; rung 3
LD W461.14  ; PB.PIN UP
LD W478.07  ; UNIT1 HOME POS.
AND H13.00  ; MB ROTATE : FINISH
ORLD
LD W478.15  ; PB all unit home
AND H13.00  ; MB ROTATE : FINISH
ORLD
ANDNOT W461.15  ; PB.PIN DOWN
LD PH_3304_08_ON  ; PH. WORK ROTATE PRE-END CONFIRM on
OR GSB000  ; FOR EQUIPMENT DESIGN_ORDINARY TIMES ON
ANDLD
ANDNOT LS_3303_08  ; AS.PIN POSIRIONNING UP CONFIRM
OUT W55.14  ; IND.PIN UP
; rung 4
LD W461.15  ; PB.PIN DOWN
LD W478.15  ; PB all unit home
OR W478.07  ; UNIT1 HOME POS.
ANDNOT H13.00  ; MB ROTATE : FINISH
ORLD
ANDNOT W461.14  ; PB.PIN UP
LDNOT H12.00  ; Vacum work memory
OR GSB000  ; FOR EQUIPMENT DESIGN_ORDINARY TIMES ON
ANDLD
LD PH_3302_15_OFF  ; PH. WORK IN ROTATE UNIT CONFIRM off
OR GSB000  ; FOR EQUIPMENT DESIGN_ORDINARY TIMES ON
ANDLD
AND LS_3303_05  ; AS.M&B LOAD OUT UNIT UP.CONFIRM
LD PH_3304_08_OFF  ; PH. WORK ROTATE PRE-END CONFIRM off
AND PH_3304_09_OFF  ; PH. TEMINAL IN POSITION CONFIRM off
OR GSB000  ; FOR EQUIPMENT DESIGN_ORDINARY TIMES ON
ANDLD
ANDNOT LS_3303_09  ; AS.PIN POSIRIONNING DOWN CONFIRM
OUT W55.15  ; PB.PIN DOWN
; rung 5
ILC(003)

### Section END
; rung 0
END(001)

## Program P13_DIAPH_SHUTTER (cyclic task 3)
Local symbols
LB11400 E0_43.01 BOOL  ; Auto start begin
LB11401 E0_43.02 BOOL  ; door Enable
LB11402 E0_43.03 BOOL  ; enable confirm
LB11403 E0_43.05 BOOL  ; Shutter 2 down
LB11404 E0_43.04 BOOL  ; SHUTTER DOOR 2 DOWN CONF
LB11407 E0_43.06 BOOL  ; Door enable
LB11408 E0_43.07 BOOL  ; door enable conf
LB11409 E0_43.08 BOOL  ; shutter 2 up
LB11410 E0_43.09 BOOL  ; shutter 2 up conf
LB11599 E0_43.10 BOOL  ; p13 _1 cycle end
LB1300 E0_43.11 BOOL  ; P13_2 cycle start
LB1301 E0_43.00 BOOL  ; COVER 2 close
LB1303 E0_14.00 BOOL  ; Cover 2 Open
LB1400 E0_14.01 BOOL  ; AUTO START BEGIN
LB1401 E0_14.02 BOOL  ; DIAPHAM DOOR ENABLE
LB1402 E0_14.03 BOOL  ; DIAPHAM DOOR ENABLE CONF
LB1403 E0_14.04 BOOL  ; SHUTTER DOOR 1 DOWN
LB1404 E0_14.05 BOOL  ; SHUTTER DOOR 1 DOWN CONF
LB1405 E0_14.06 BOOL  ; SHUTTER DOOR 2 UP
LB1406 E0_14.07 BOOL  ; SHUTTER DOOR 2 UP
LB1407 E0_14.08 BOOL  ; DIAPHAM DOOR ENABLE
LB1408 E0_14.09 BOOL  ; DIAPHAM DOOR ENABLE CONF
LB1409 E0_14.10 BOOL  ; SHUTTER DOOR 1 UP
LB1410 E0_14.11 BOOL  ; SHUTTER DOOR 1 UP CONf
LB1411 E0_14.12 BOOL  ; SHUTTER DOOR 2 DOWN
LB1412 E0_14.13 BOOL  ; SHUTTER DOOR 2 DOWN CONF
LB1413 E0_14.14 BOOL  ; AUTO START BEGIN
LB1414 E0_14.15 BOOL  ; DIAPHAM DOOR ENABLE
LB1415 E0_15.00 BOOL  ; DIAPHAM DOOR ENABLE CONF
LB1416 E0_15.01 BOOL  ; SHUTTER DOOR 1 DOWN
LB1417 E0_15.02 BOOL  ; SHUTTER DOOR 1 DOWN
LB1418 E0_15.03 BOOL  ; SHUTTER DOOR 2 UP
LB1419 E0_15.04 BOOL  ; SHUTTER DOOR 2 UP CONF
LB1420 E0_15.05 BOOL  ; DIAPHAM DOOR ENABLE
LB1421 E0_15.06 BOOL  ; DIAPHAM DOOR ENABLE CONF
LB1422 E0_15.07 BOOL  ; SHUTTER DOOR 1 UP
LB1423 E0_15.08 BOOL  ; SHUTTER DOOR 1 UP CONF
LB1424 E0_15.09 BOOL  ; SHUTTER DOOR 2 DOWN
LB1425 E0_15.10 BOOL  ; SHUTTER DOOR 2 DOWN CONF
LB1450 E0_45.09 BOOL  ; ind 1 cycle p13a
LB1599 E0_15.11 BOOL  ; P13 AutoCycleEnd
LB300 E0_15.12 BOOL  ; P13 CycleStart
LB301 E0_15.13 BOOL  ; P13 shutter 1 close condition
LB302 E0_15.14 BOOL  ; P13 case2
LB303 E0_15.15 BOOL  ; P13 shutter 1 open cond
LB4312 E0_46.01 BOOL
LB75091 E0_43.12 BOOL  ; p13a motion start
LB9209 E0_43.14 BOOL  ; P13a motion cond
LB93 E0_42.14 BOOL  ; Shutter 2 Close cond
LB94 E0_42.15 BOOL  ; SHUtter 2 Open cond
LT1432 T3036 TIMER
LT3431 T3018 TIMER
LT432 T3019 TIMER
LT529 T3040 TIMER
LT657 T3039 TIMER
hgb E0_45.08 BOOL
mem_IND_Down E0_16.00 BOOL

### Section HMI_Output

### Section Autorun

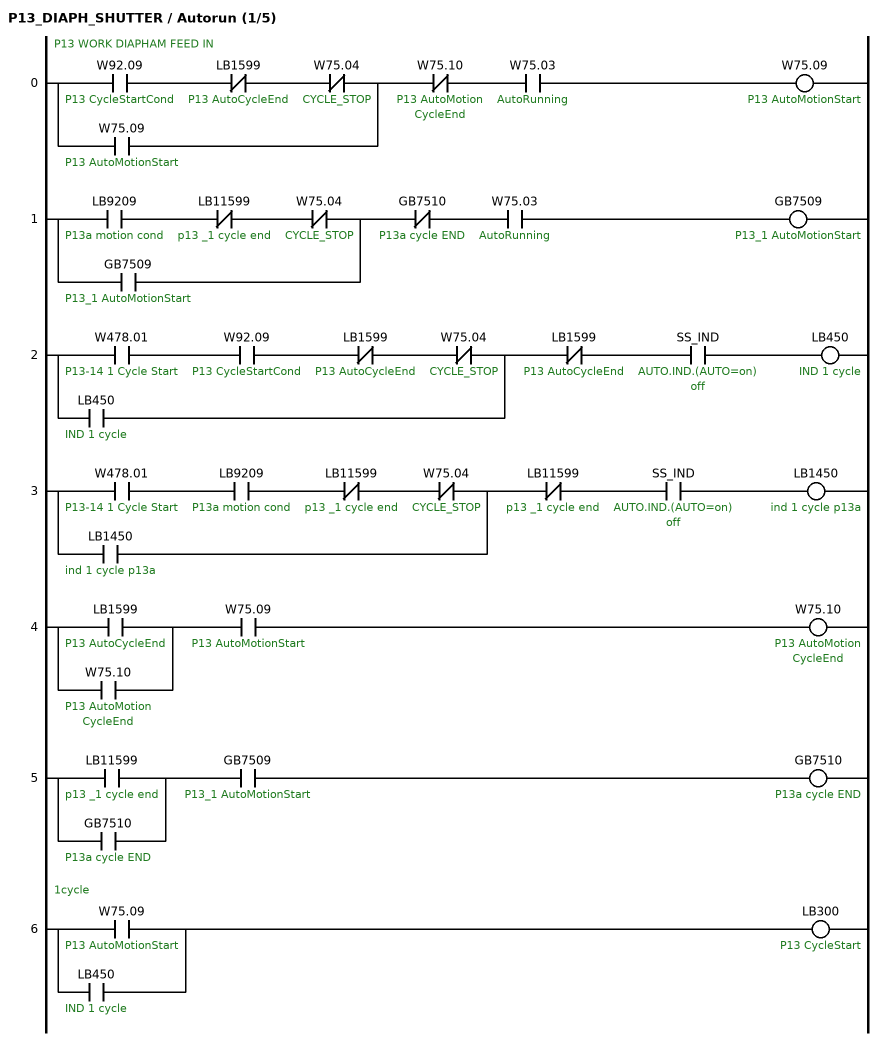
; rung 0: P13 WORK DIAPHAM FEED IN
LD W92.09  ; P13 CycleStartCond
ANDNOT LB1599  ; P13 AutoCycleEnd
ANDNOT W75.04  ; CYCLE_STOP
OR W75.09  ; P13 AutoMotionStart
ANDNOT W75.10  ; P13 AutoMotion CycleEnd
AND W75.03  ; AutoRunning
OUT W75.09  ; P13 AutoMotionStart
; rung 1
LD LB9209  ; P13a motion cond
ANDNOT LB11599  ; p13 _1 cycle end
ANDNOT W75.04  ; CYCLE_STOP
OR GB7509  ; P13_1 AutoMotionStart
ANDNOT GB7510  ; P13a cycle END
AND W75.03  ; AutoRunning
OUT GB7509  ; P13_1 AutoMotionStart
; rung 2
LD W478.01  ; P13-14 1 Cycle Start
AND W92.09  ; P13 CycleStartCond
ANDNOT LB1599  ; P13 AutoCycleEnd
ANDNOT W75.04  ; CYCLE_STOP
OR LB450  ; IND 1 cycle
ANDNOT LB1599  ; P13 AutoCycleEnd
AND SS_IND  ; AUTO.IND.(AUTO=on) off
OUT LB450  ; IND 1 cycle
; rung 3
LD W478.01  ; P13-14 1 Cycle Start
AND LB9209  ; P13a motion cond
ANDNOT LB11599  ; p13 _1 cycle end
ANDNOT W75.04  ; CYCLE_STOP
OR LB1450  ; ind 1 cycle p13a
ANDNOT LB11599  ; p13 _1 cycle end
AND SS_IND  ; AUTO.IND.(AUTO=on) off
OUT LB1450  ; ind 1 cycle p13a
; rung 4
LD LB1599  ; P13 AutoCycleEnd
OR W75.10  ; P13 AutoMotion CycleEnd
AND W75.09  ; P13 AutoMotionStart
OUT W75.10  ; P13 AutoMotion CycleEnd
; rung 5
LD LB11599  ; p13 _1 cycle end
OR GB7510  ; P13a cycle END
AND GB7509  ; P13_1 AutoMotionStart
OUT GB7510  ; P13a cycle END
; rung 6: 1cycle
LD W75.09  ; P13 AutoMotionStart
OR LB450  ; IND 1 cycle
OUT LB300  ; P13 CycleStart

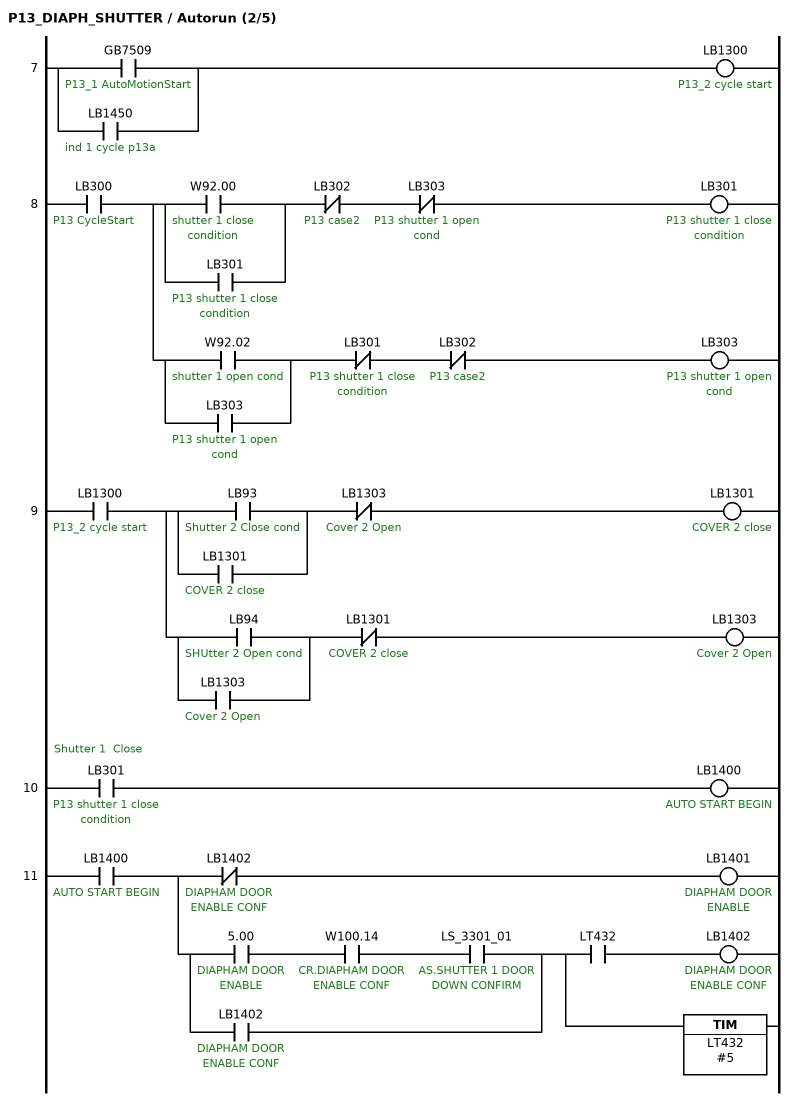
; rung 7
LD GB7509  ; P13_1 AutoMotionStart
OR LB1450  ; ind 1 cycle p13a
OUT LB1300  ; P13_2 cycle start
; rung 8
LD LB300  ; P13 CycleStart
OUT TR0
LD W92.00  ; shutter 1 close condition
OR LB301  ; P13 shutter 1 close condition
ANDLD
ANDNOT LB302  ; P13 case2
ANDNOT LB303  ; P13 shutter 1 open cond
OUT LB301  ; P13 shutter 1 close condition
LD TR0
LD W92.02  ; shutter 1 open cond
OR LB303  ; P13 shutter 1 open cond
ANDLD
ANDNOT LB301  ; P13 shutter 1 close condition
ANDNOT LB302  ; P13 case2
OUT LB303  ; P13 shutter 1 open cond
; rung 9
LD LB1300  ; P13_2 cycle start
OUT TR0
LD LB93  ; Shutter 2 Close cond
OR LB1301  ; COVER 2 close
ANDLD
ANDNOT LB1303  ; Cover 2 Open
OUT LB1301  ; COVER 2 close
LD TR0
LD LB94  ; SHUtter 2 Open cond
OR LB1303  ; Cover 2 Open
ANDLD
ANDNOT LB1301  ; COVER 2 close
OUT LB1303  ; Cover 2 Open
; rung 10: Shutter 1  Close
LD LB301  ; P13 shutter 1 close condition
OUT LB1400  ; AUTO START BEGIN
; rung 11
LD LB1400  ; AUTO START BEGIN
OUT TR0
ANDNOT LB1402  ; DIAPHAM DOOR ENABLE CONF
OUT LB1401  ; DIAPHAM DOOR ENABLE
LD TR0
LD 5.00  ; DIAPHAM DOOR ENABLE
AND W100.14  ; CR.DIAPHAM DOOR ENABLE CONF
AND LS_3301_01  ; AS.SHUTTER 1 DOOR DOWN CONFIRM
OR LB1402  ; DIAPHAM DOOR ENABLE CONF
ANDLD
OUT TR0
AND LT432
OUT LB1402  ; DIAPHAM DOOR ENABLE CONF
LD TR0
TIM LT432 #5

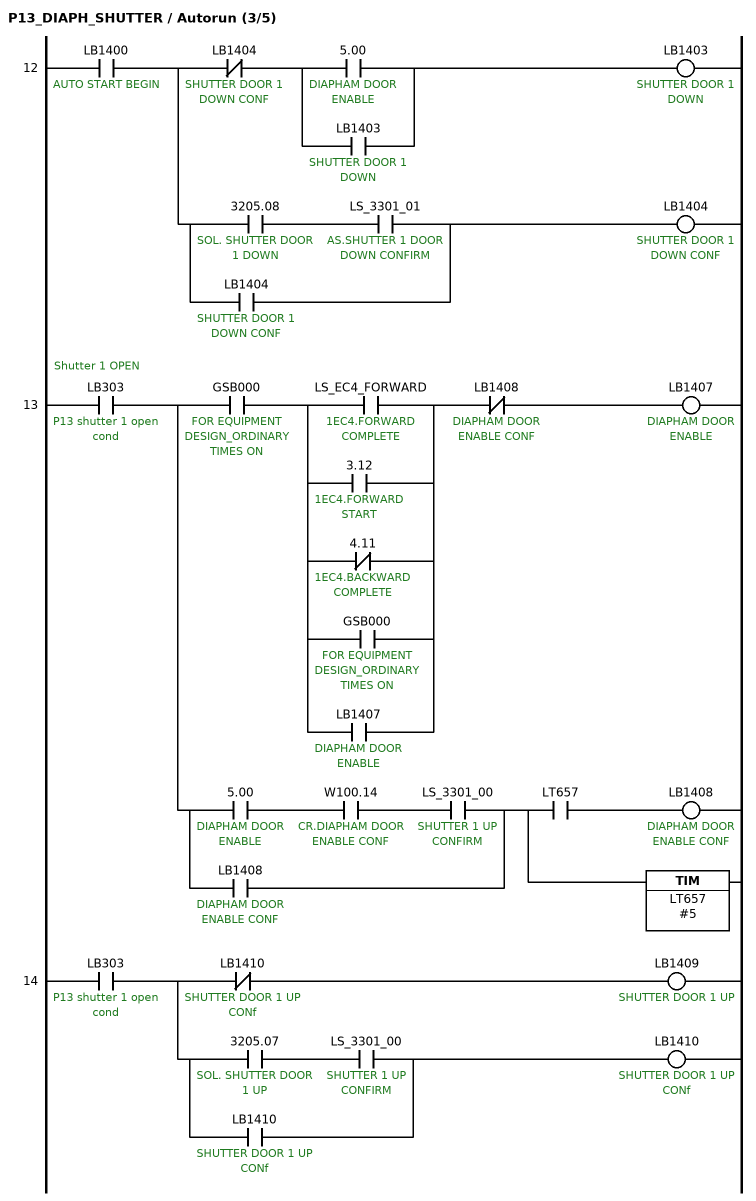
; rung 12
LD LB1400  ; AUTO START BEGIN
OUT TR0
ANDNOT LB1404  ; SHUTTER DOOR 1 DOWN CONF
LD 5.00  ; DIAPHAM DOOR ENABLE
OR LB1403  ; SHUTTER DOOR 1 DOWN
ANDLD
OUT LB1403  ; SHUTTER DOOR 1 DOWN
LD TR0
LD 3205.08  ; SOL. SHUTTER DOOR 1 DOWN
AND LS_3301_01  ; AS.SHUTTER 1 DOOR DOWN CONFIRM
OR LB1404  ; SHUTTER DOOR 1 DOWN CONF
ANDLD
OUT LB1404  ; SHUTTER DOOR 1 DOWN CONF
; rung 13: Shutter 1 OPEN
LD LB303  ; P13 shutter 1 open cond
OUT TR0
AND GSB000  ; FOR EQUIPMENT DESIGN_ORDINARY TIMES ON
LD LS_EC4_FORWARD  ; 1EC4.FORWARD COMPLETE
OR 3.12  ; 1EC4.FORWARD START
ORNOT 4.11  ; 1EC4.BACKWARD COMPLETE
OR GSB000  ; FOR EQUIPMENT DESIGN_ORDINARY TIMES ON
OR LB1407  ; DIAPHAM DOOR ENABLE
ANDLD
ANDNOT LB1408  ; DIAPHAM DOOR ENABLE CONF
OUT LB1407  ; DIAPHAM DOOR ENABLE
LD TR0
LD 5.00  ; DIAPHAM DOOR ENABLE
AND W100.14  ; CR.DIAPHAM DOOR ENABLE CONF
AND LS_3301_00  ; SHUTTER 1 UP CONFIRM
OR LB1408  ; DIAPHAM DOOR ENABLE CONF
ANDLD
OUT TR0
AND LT657
OUT LB1408  ; DIAPHAM DOOR ENABLE CONF
LD TR0
TIM LT657 #5
; rung 14
LD LB303  ; P13 shutter 1 open cond
OUT TR0
ANDNOT LB1410  ; SHUTTER DOOR 1 UP CONf
OUT LB1409  ; SHUTTER DOOR 1 UP
LD TR0
LD 3205.07  ; SOL. SHUTTER DOOR 1 UP
AND LS_3301_00  ; SHUTTER 1 UP CONFIRM
OR LB1410  ; SHUTTER DOOR 1 UP CONf
ANDLD
OUT LB1410  ; SHUTTER DOOR 1 UP CONf

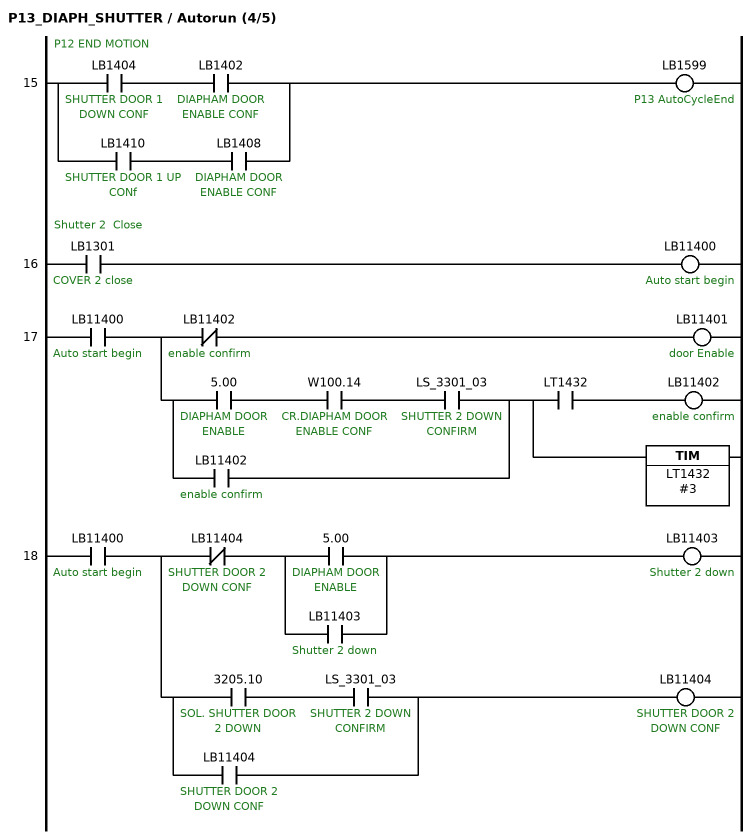
; rung 15: P12 END MOTION
LD LB1404  ; SHUTTER DOOR 1 DOWN CONF
AND LB1402  ; DIAPHAM DOOR ENABLE CONF
LD LB1410  ; SHUTTER DOOR 1 UP CONf
AND LB1408  ; DIAPHAM DOOR ENABLE CONF
ORLD
OUT LB1599  ; P13 AutoCycleEnd
; rung 16: Shutter 2  Close
LD LB1301  ; COVER 2 close
OUT LB11400  ; Auto start begin
; rung 17
LD LB11400  ; Auto start begin
OUT TR0
ANDNOT LB11402  ; enable confirm
OUT LB11401  ; door Enable
LD TR0
LD 5.00  ; DIAPHAM DOOR ENABLE
AND W100.14  ; CR.DIAPHAM DOOR ENABLE CONF
AND LS_3301_03  ; SHUTTER 2 DOWN CONFIRM
OR LB11402  ; enable confirm
ANDLD
OUT TR0
AND LT1432
OUT LB11402  ; enable confirm
LD TR0
TIM LT1432 #3
; rung 18
LD LB11400  ; Auto start begin
OUT TR0
ANDNOT LB11404  ; SHUTTER DOOR 2 DOWN CONF
LD 5.00  ; DIAPHAM DOOR ENABLE
OR LB11403  ; Shutter 2 down
ANDLD
OUT LB11403  ; Shutter 2 down
LD TR0
LD 3205.10  ; SOL. SHUTTER DOOR 2 DOWN
AND LS_3301_03  ; SHUTTER 2 DOWN CONFIRM
OR LB11404  ; SHUTTER DOOR 2 DOWN CONF
ANDLD
OUT LB11404  ; SHUTTER DOOR 2 DOWN CONF

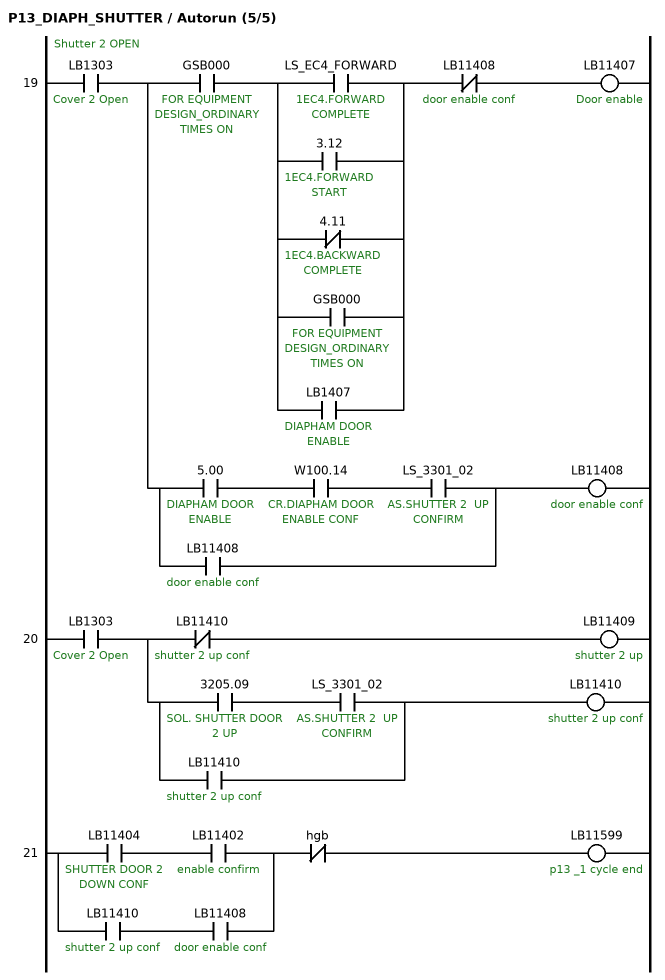
; rung 19: Shutter 2 OPEN
LD LB1303  ; Cover 2 Open
OUT TR0
AND GSB000  ; FOR EQUIPMENT DESIGN_ORDINARY TIMES ON
LD LS_EC4_FORWARD  ; 1EC4.FORWARD COMPLETE
OR 3.12  ; 1EC4.FORWARD START
ORNOT 4.11  ; 1EC4.BACKWARD COMPLETE
OR GSB000  ; FOR EQUIPMENT DESIGN_ORDINARY TIMES ON
OR LB1407  ; DIAPHAM DOOR ENABLE
ANDLD
ANDNOT LB11408  ; door enable conf
OUT LB11407  ; Door enable
LD TR0
LD 5.00  ; DIAPHAM DOOR ENABLE
AND W100.14  ; CR.DIAPHAM DOOR ENABLE CONF
AND LS_3301_02  ; AS.SHUTTER 2  UP CONFIRM
OR LB11408  ; door enable conf
ANDLD
OUT LB11408  ; door enable conf
; rung 20
LD LB1303  ; Cover 2 Open
OUT TR0
ANDNOT LB11410  ; shutter 2 up conf
OUT LB11409  ; shutter 2 up
LD TR0
LD 3205.09  ; SOL. SHUTTER DOOR 2 UP
AND LS_3301_02  ; AS.SHUTTER 2  UP CONFIRM
OR LB11410  ; shutter 2 up conf
ANDLD
OUT LB11410  ; shutter 2 up conf
; rung 21
LD LB11404  ; SHUTTER DOOR 2 DOWN CONF
AND LB11402  ; enable confirm
LD LB11410  ; shutter 2 up conf
AND LB11408  ; door enable conf
ORLD
ANDNOT hgb
OUT LB11599  ; p13 _1 cycle end

### Section Condition

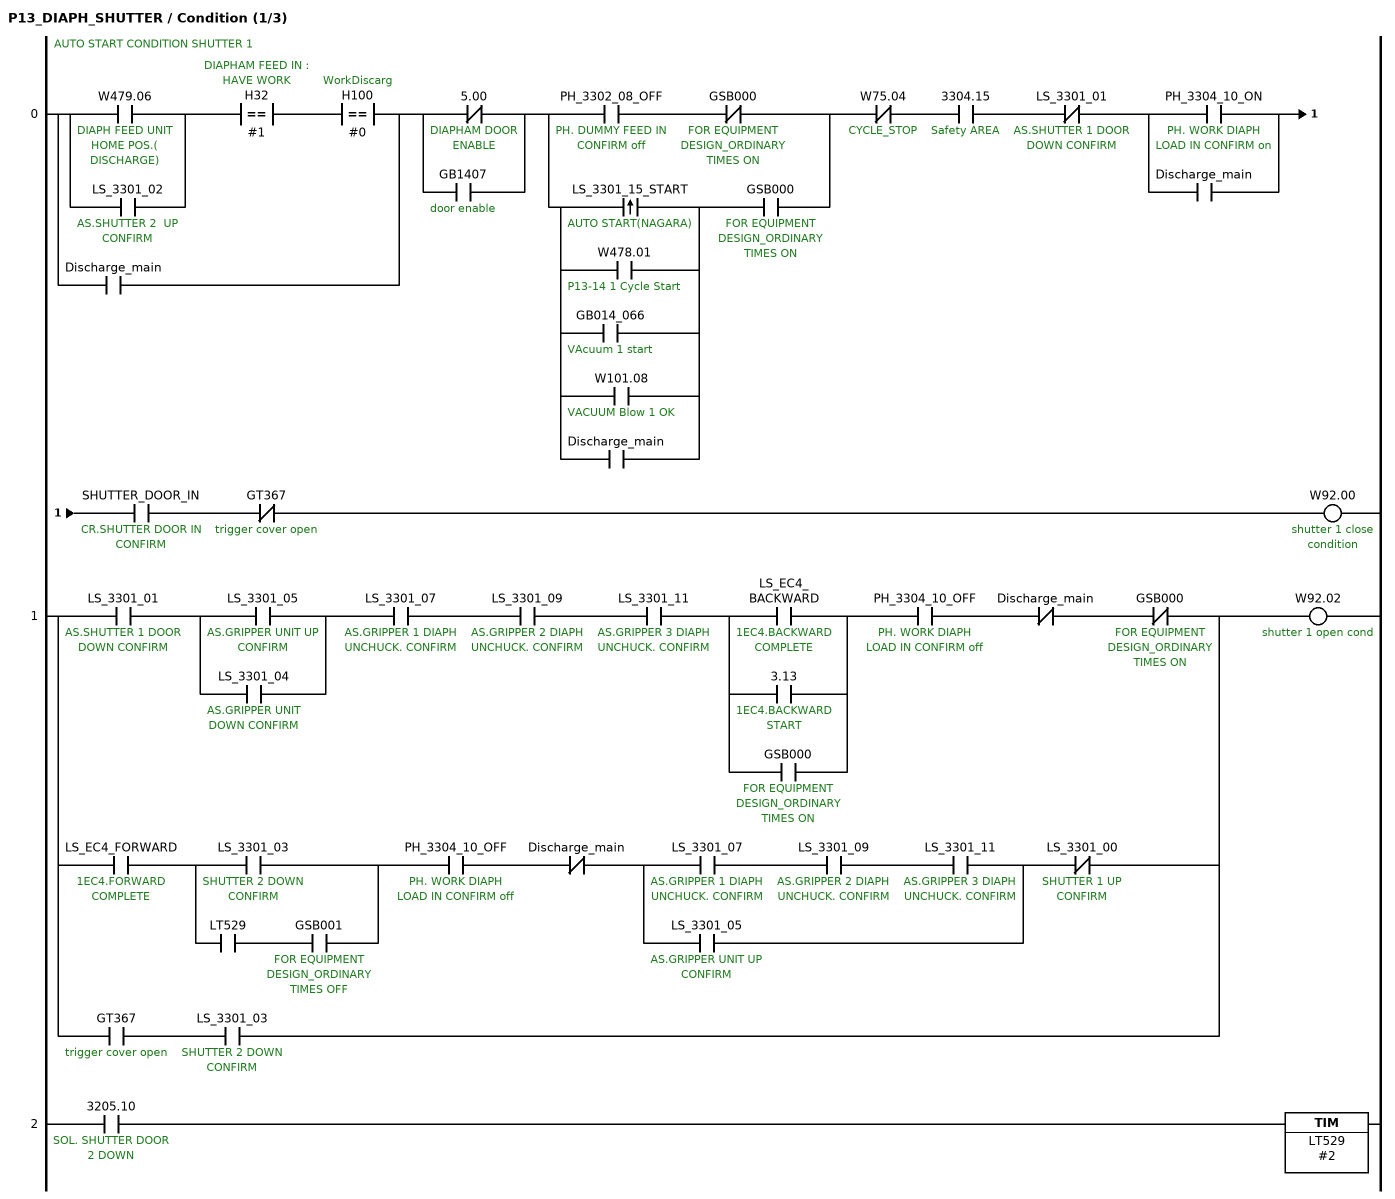
; rung 0: AUTO START CONDITION SHUTTER 1
LD W479.06  ; DIAPH FEED UNIT HOME POS.(DISCHARGE)
OR LS_3301_02  ; AS.SHUTTER 2  UP CONFIRM
AND=(300) H32 #1  ; DIAPHAM FEED IN : HAVE WORK
AND=(300) H100 #0  ; WorkDiscarg
OR Discharge_main
LDNOT 5.00  ; DIAPHAM DOOR ENABLE
OR GB1407  ; door enable
ANDLD
LD PH_3302_08_OFF  ; PH. DUMMY FEED IN CONFIRM off
ANDNOT GSB000  ; FOR EQUIPMENT DESIGN_ORDINARY TIMES ON
@LD LS_3301_15_START  ; AUTO START(NAGARA)
OR W478.01  ; P13-14 1 Cycle Start
OR GB014_066  ; VAcuum 1 start
OR W101.08  ; VACUUM Blow 1 OK
OR Discharge_main
AND GSB000  ; FOR EQUIPMENT DESIGN_ORDINARY TIMES ON
ORLD
ANDLD
ANDNOT W75.04  ; CYCLE_STOP
AND 3304.15  ; Safety AREA
ANDNOT LS_3301_01  ; AS.SHUTTER 1 DOOR DOWN CONFIRM
LD PH_3304_10_ON  ; PH. WORK DIAPH LOAD IN CONFIRM on
OR Discharge_main
ANDLD
AND SHUTTER_DOOR_IN  ; CR.SHUTTER DOOR IN CONFIRM
ANDNOT GT367  ; trigger cover open
OUT W92.00  ; shutter 1 close condition
; rung 1
LD LS_3301_01  ; AS.SHUTTER 1 DOOR DOWN CONFIRM
LD LS_3301_05  ; AS.GRIPPER UNIT UP CONFIRM
OR LS_3301_04  ; AS.GRIPPER UNIT DOWN CONFIRM
ANDLD
AND LS_3301_07  ; AS.GRIPPER 1 DIAPH UNCHUCK. CONFIRM
AND LS_3301_09  ; AS.GRIPPER 2 DIAPH UNCHUCK. CONFIRM
AND LS_3301_11  ; AS.GRIPPER 3 DIAPH UNCHUCK. CONFIRM
LD LS_EC4_BACKWARD  ; 1EC4.BACKWARD COMPLETE
OR 3.13  ; 1EC4.BACKWARD START
OR GSB000  ; FOR EQUIPMENT DESIGN_ORDINARY TIMES ON
ANDLD
AND PH_3304_10_OFF  ; PH. WORK DIAPH LOAD IN CONFIRM off
ANDNOT Discharge_main
ANDNOT GSB000  ; FOR EQUIPMENT DESIGN_ORDINARY TIMES ON
LD LS_EC4_FORWARD  ; 1EC4.FORWARD COMPLETE
LD LS_3301_03  ; SHUTTER 2 DOWN CONFIRM
LD LT529
AND GSB001  ; FOR EQUIPMENT DESIGN_ORDINARY TIMES OFF
ORLD
ANDLD
AND PH_3304_10_OFF  ; PH. WORK DIAPH LOAD IN CONFIRM off
ANDNOT Discharge_main
LD LS_3301_07  ; AS.GRIPPER 1 DIAPH UNCHUCK. CONFIRM
AND LS_3301_09  ; AS.GRIPPER 2 DIAPH UNCHUCK. CONFIRM
AND LS_3301_11  ; AS.GRIPPER 3 DIAPH UNCHUCK. CONFIRM
OR LS_3301_05  ; AS.GRIPPER UNIT UP CONFIRM
ANDLD
ANDNOT LS_3301_00  ; SHUTTER 1 UP CONFIRM
ORLD
LD GT367  ; trigger cover open
AND LS_3301_03  ; SHUTTER 2 DOWN CONFIRM
ORLD
OUT W92.02  ; shutter 1 open cond
; rung 2
LD 3205.10  ; SOL. SHUTTER DOOR 2 DOWN
TIM LT529 #2

